LIN {X 0,Y 114.855,Z 265.173,A -85,B 0,C 180,E1 -25888.942,E2 -25888.942} C_VEL
LIN {X 0,Y 114.946,Z 265.116,A -85,B 0,C 180,E1 -25896.507,E2 -25896.507} C_VEL
LIN {X 0,Y 115.013,Z 265.157,A -85,B 0,C 180,E1 -25902.21,E2 -25902.21} C_VEL
LIN {X 0,Y 115.285,Z 265.077,A -85,B 0,C 180,E1 -25907.258,E2 -25907.258} C_VEL
LIN {X 0,Y 115.397,Z 265.09,A -85,B 0,C 180,E1 -25913.003,E2 -25913.003} C_VEL
LIN {X 0,Y 115.994,Z 264.995,A -85,B 0,C 180,E1 -25920,E2 -25920} C_VEL
LIN {X 0,Y 115.392,Z 265.108,A -85,B 0,C 180,E1 -25926.996,E2 -25926.996} C_VEL
LIN {X 0,Y 115.284,Z 265.085,A -85,B 0,C 180,E1 -25932.739,E2 -25932.739} C_VEL
LIN {X 0,Y 114.998,Z 265.157,A -85,B 0,C 180,E1 -25939.525,E2 -25939.525} C_VEL
LIN {X 0,Y 115.938,Z 267.926,A -85,B 0,C 180,E1 -25940.747,E2 -25940.747} C_VEL
LIN {X 0,Y 117.848,Z 270.02,A -85,B 0,C 180,E1 -25942.524,E2 -25942.524} C_VEL
LIN {X 0,Y 119.053,Z 270.961,A -85,B 0,C 180,E1 -25943.531,E2 -25943.531} C_VEL
LIN {X 0,Y 120.863,Z 274.022,A -85,B 0,C 180,E1 -25945.164,E2 -25945.164} C_VEL
LIN {X 0,Y 122.793,Z 276.078,A -85,B 0,C 180,E1 -25946.675,E2 -25946.675} C_VEL
LIN {X 0,Y 125.302,Z 279.71,A -85,B 0,C 180,E1 -25948.59,E2 -25948.59} C_VEL
LIN {X 0,Y 129.507,Z 285.851,A -85,B 0,C 180,E1 -25951.488,E2 -25951.488} C_VEL
LIN {X 0,Y 134.666,Z 293.955,A -85,B 0,C 180,E1 -25954.693,E2 -25954.693} C_VEL
LIN {X 0,Y 138.207,Z 301.272,A -85,B 0,C 180,E1 -25956.805,E2 -25956.805} C_VEL
LIN {X 0,Y 143.082,Z 312.975,A -85,B 0,C 180,E1 -25959.569,E2 -25959.569} C_VEL
LIN {X 0,Y 147.64,Z 326.29,A -85,B 0,C 180,E1 -25962.08,E2 -25962.08} C_VEL
LIN {X 0,Y 144.395,Z 368.364,A -85,B 0,C 180,E1 -25963.988,E2 -25963.988} C_VEL
LIN {X 0,Y 142.249,Z 381.813,A -85,B 0,C 180,E1 -25965.008,E2 -25965.008} C_VEL
LIN {X 0,Y 139.648,Z 394.07,A -85,B 0,C 180,E1 -25966.462,E2 -25966.462} C_VEL
LIN {X 0,Y 136.244,Z 405.888,A -85,B 0,C 180,E1 -25968.385,E2 -25968.385} C_VEL
LIN {X 0,Y 132.886,Z 416.032,A -85,B 0,C 180,E1 -25970.607,E2 -25970.607} C_VEL
LIN {X 0,Y 128.827,Z 426.583,A -85,B 0,C 180,E1 -25973.611,E2 -25973.611} C_VEL
LIN {X 0,Y 125.2,Z 435.221,A -85,B 0,C 180,E1 -25976.819,E2 -25976.819} C_VEL
LIN {X 0,Y 121.652,Z 443.346,A -85,B 0,C 180,E1 -25980.697,E2 -25980.697} C_VEL
LIN {X 0,Y 118.219,Z 450.929,A -85,B 0,C 180,E1 -25985.41,E2 -25985.41} C_VEL
LIN {X 0,Y 115.387,Z 457.118,A -85,B 0,C 180,E1 -25990.429,E2 -25990.429} C_VEL
LIN {X 0,Y 113.579,Z 462.024,A -85,B 0,C 180,E1 -25995.67,E2 -25995.67} C_VEL
LIN {X 0,Y 112.543,Z 465.767,A -85,B 0,C 180,E1 -26001.019,E2 -26001.019} C_VEL
LIN {X 0,Y 112.201,Z 468.455,A -85,B 0,C 180,E1 -26006.409,E2 -26006.409} C_VEL
LIN {X 0,Y 112.263,Z 469.704,A -85,B 0,C 180,E1 -26010.001,E2 -26010.001} C_VEL
LIN {X 0,Y 112.2,Z 470.534,A -85,B 0,C 180,E1 -26013.592,E2 -26013.592} C_VEL
LIN {X 0,Y 112.334,Z 470.932,A -85,B 0,C 180,E1 -26017.189,E2 -26017.189} C_VEL
LIN {X 0,Y 113.649,Z 470.568,A -85,B 0,C 180,E1 -26024.322,E2 -26024.322} C_VEL
LIN {X 0,Y 116.47,Z 468.695,A -85,B 0,C 180,E1 -26031.227,E2 -26031.227} C_VEL
LIN {X 0,Y 121.115,Z 465.171,A -85,B 0,C 180,E1 -26037.66,E2 -26037.66} C_VEL
LIN {X 0,Y 125.472,Z 461.407,A -85,B 0,C 180,E1 -26042.149,E2 -26042.149} C_VEL
LIN {X 0,Y 130.501,Z 456.57,A -85,B 0,C 180,E1 -26046.327,E2 -26046.327} C_VEL
LIN {X 0,Y 137.171,Z 449.407,A -85,B 0,C 180,E1 -26050.787,E2 -26050.787} C_VEL
LIN {X 0,Y 143.707,Z 441.626,A -85,B 0,C 180,E1 -26054.179,E2 -26054.179} C_VEL
LIN {X 0,Y 150.624,Z 432.012,A -85,B 0,C 180,E1 -26057.298,E2 -26057.298} C_VEL
LIN {X 0,Y 156.829,Z 422.095,A -85,B 0,C 180,E1 -26059.625,E2 -26059.625} C_VEL
LIN {X 0,Y 159.223,Z 417.796,A -85,B 0,C 180,E1 -26060.431,E2 -26060.431} C_VEL
LIN {X 0,Y 161.357,Z 413.071,A -85,B 0,C 180,E1 -26061.461,E2 -26061.461} C_VEL
LIN {X 0,Y 163.563,Z 405.279,A -85,B 0,C 180,E1 -26063.505,E2 -26063.505} C_VEL
LIN {X 0,Y 165.482,Z 397.087,A -85,B 0,C 180,E1 -26065.314,E2 -26065.314} C_VEL
LIN {X 0,Y 167.06,Z 391.752,A -85,B 0,C 180,E1 -26065.968,E2 -26065.968} C_VEL
LIN {X 0,Y 170.943,Z 378.184,A -85,B 0,C 180,E1 -26066.933,E2 -26066.933} C_VEL
LIN {X 0,Y 173.358,Z 365.954,A -85,B 0,C 180,E1 -26067.492,E2 -26067.492} C_VEL
LIN {X 0,Y 175.241,Z 348.208,A -85,B 0,C 180,E1 -26068.166,E2 -26068.166} C_VEL
LIN {X 0,Y 173.221,Z 341.92,A -85,B 0,C 180,E1 -26070.659,E2 -26070.659} C_VEL
LIN {X 0,Y 171.373,Z 336.851,A -85,B 0,C 180,E1 -26073.277,E2 -26073.277} C_VEL
LIN {X 0,Y 169.812,Z 332.855,A -85,B 0,C 180,E1 -26075.909,E2 -26075.909} C_VEL
LIN {X 0,Y 168.758,Z 330.738,A -85,B 0,C 180,E1 -26077.988,E2 -26077.988} C_VEL
LIN {X 0,Y 167.065,Z 326.954,A -85,B 0,C 180,E1 -26083.227,E2 -26083.227} C_VEL
LIN {X 0,Y 166.739,Z 326.515,A -85,B 0,C 180,E1 -26090.294,E2 -26090.294} C_VEL
LIN {X 0,Y 167.542,Z 327.166,A -85,B 0,C 180,E1 -26093.868,E2 -26093.868} C_VEL
LIN {X 0,Y 169.247,Z 331.048,A -85,B 0,C 180,E1 -26098.353,E2 -26098.353} C_VEL
LIN {X 0,Y 171.178,Z 334.972,A -85,B 0,C 180,E1 -26101.648,E2 -26101.648} C_VEL
LIN {X 0,Y 173.938,Z 340.804,A -85,B 0,C 180,E1 -26105.301,E2 -26105.301} C_VEL
LIN {X 0,Y 175.586,Z 344.85,A -85,B 0,C 180,E1 -26107.174,E2 -26107.174} C_VEL
LIN {X 0,Y 173.207,Z 364.688,A -85,B 0,C 180,E1 -26107.837,E2 -26107.837} C_VEL
LIN {X 0,Y 170.577,Z 377.505,A -85,B 0,C 180,E1 -26108.571,E2 -26108.571} C_VEL
LIN {X 0,Y 166.926,Z 389.808,A -85,B 0,C 180,E1 -26109.597,E2 -26109.597} C_VEL
LIN {X 0,Y 162.787,Z 400.561,A -85,B 0,C 180,E1 -26110.831,E2 -26110.831} C_VEL
LIN {X 0,Y 157.521,Z 411.598,A -85,B 0,C 180,E1 -26112.516,E2 -26112.516} C_VEL
LIN {X 0,Y 151.614,Z 421.914,A -85,B 0,C 180,E1 -26114.614,E2 -26114.614} C_VEL
LIN {X 0,Y 145.495,Z 430.892,A -85,B 0,C 180,E1 -26117.028,E2 -26117.028} C_VEL
LIN {X 0,Y 138.67,Z 439.441,A -85,B 0,C 180,E1 -26120.118,E2 -26120.118} C_VEL
LIN {X 0,Y 132.225,Z 446.432,A -85,B 0,C 180,E1 -26123.528,E2 -26123.528} C_VEL
LIN {X 0,Y 126.447,Z 451.978,A -85,B 0,C 180,E1 -26127.216,E2 -26127.216} C_VEL
LIN {X 0,Y 120.926,Z 456.69,A -85,B 0,C 180,E1 -26131.538,E2 -26131.538} C_VEL
LIN {X 0,Y 114.755,Z 461.213,A -85,B 0,C 180,E1 -26137.766,E2 -26137.766} C_VEL
LIN {X 0,Y 110.03,Z 464.019,A -85,B 0,C 180,E1 -26144.637,E2 -26144.637} C_VEL
LIN {X 0,Y 106.69,Z 465.22,A -85,B 0,C 180,E1 -26152.231,E2 -26152.231} C_VEL
LIN {X 0,Y 105.248,Z 465.079,A -85,B 0,C 180,E1 -26157.71,E2 -26157.71} C_VEL
LIN {X 0,Y 104.725,Z 464.378,A -85,B 0,C 180,E1 -26161.981,E2 -26161.981} C_VEL
LIN {X 0,Y 104.598,Z 463.238,A -85,B 0,C 180,E1 -26166.225,E2 -26166.225} C_VEL
LIN {X 0,Y 105.233,Z 460.602,A -85,B 0,C 180,E1 -26172.51,E2 -26172.51} C_VEL
LIN {X 0,Y 106.709,Z 456.837,A -85,B 0,C 180,E1 -26178.604,E2 -26178.604} C_VEL
LIN {X 0,Y 108.848,Z 451.866,A -85,B 0,C 180,E1 -26184.442,E2 -26184.442} C_VEL
LIN {X 0,Y 111.866,Z 445.532,A -85,B 0,C 180,E1 -26189.999,E2 -26189.999} C_VEL
LIN {X 0,Y 115.781,Z 437.599,A -85,B 0,C 180,E1 -26195.224,E2 -26195.224} C_VEL
LIN {X 0,Y 119.644,Z 429.439,A -85,B 0,C 180,E1 -26199.296,E2 -26199.296} C_VEL
LIN {X 0,Y 123.956,Z 419.414,A -85,B 0,C 180,E1 -26203.108,E2 -26203.108} C_VEL
LIN {X 0,Y 128.326,Z 408.2,A -85,B 0,C 180,E1 -26206.3,E2 -26206.3} C_VEL
LIN {X 0,Y 131.878,Z 397.261,A -85,B 0,C 180,E1 -26208.647,E2 -26208.647} C_VEL
LIN {X 0,Y 135.122,Z 385.083,A -85,B 0,C 180,E1 -26210.573,E2 -26210.573} C_VEL
LIN {X 0,Y 137.623,Z 372.215,A -85,B 0,C 180,E1 -26212.056,E2 -26212.056} C_VEL
LIN {X 0,Y 139.422,Z 359.052,A -85,B 0,C 180,E1 -26212.988,E2 -26212.988} C_VEL
LIN {X 0,Y 142.507,Z 321.432,A -85,B 0,C 180,E1 -26214.64,E2 -26214.64} C_VEL
LIN {X 0,Y 135.741,Z 307.538,A -85,B 0,C 180,E1 -26218.335,E2 -26218.335} C_VEL
LIN {X 0,Y 130.296,Z 297.995,A -85,B 0,C 180,E1 -26221.645,E2 -26221.645} C_VEL
LIN {X 0,Y 126.382,Z 291.705,A -85,B 0,C 180,E1 -26224.24,E2 -26224.24} C_VEL
LIN {X 0,Y 121.795,Z 284.959,A -85,B 0,C 180,E1 -26227.641,E2 -26227.641} C_VEL
LIN {X 0,Y 119.203,Z 281.373,A -85,B 0,C 180,E1 -26229.767,E2 -26229.767} C_VEL
LIN {X 0,Y 116.629,Z 278.048,A -85,B 0,C 180,E1 -26232.044,E2 -26232.044} C_VEL
LIN {X 0,Y 115.814,Z 276.758,A -85,B 0,C 180,E1 -26232.844,E2 -26232.844} C_VEL
LIN {X 0,Y 113.43,Z 274.3,A -85,B 0,C 180,E1 -26235.187,E2 -26235.187} C_VEL
LIN {X 0,Y 112.045,Z 271.721,A -85,B 0,C 180,E1 -26236.838,E2 -26236.838} C_VEL
LIN {X 0,Y 109.395,Z 269.857,A -85,B 0,C 180,E1 -26239.838,E2 -26239.838} C_VEL
LIN {X 0,Y 108.067,Z 267.583,A -85,B 0,C 180,E1 -26241.77,E2 -26241.77} C_VEL
LIN {X 0,Y 107.736,Z 266.027,A -85,B 0,C 180,E1 -26242.558,E2 -26242.558} C_VEL
LIN {X 0,Y 107.791,Z 266.049,A -85,B 0,C 180,E1 -26248.56,E2 -26248.56} C_VEL
LIN {X 0,Y 107.911,Z 265.992,A -85,B 0,C 180,E1 -26256.997,E2 -26256.997} C_VEL
LIN {X 0,Y 108.037,Z 266.005,A -85,B 0,C 180,E1 -26264.917,E2 -26264.917} C_VEL
LIN {X 0,Y 108.292,Z 265.939,A -85,B 0,C 180,E1 -26268.773,E2 -26268.773} C_VEL
LIN {X 0,Y 108.462,Z 265.973,A -85,B 0,C 180,E1 -26276.285,E2 -26276.285} C_VEL
LIN {X 0,Y 108.945,Z 265.871,A -85,B 0,C 180,E1 -26280,E2 -26280} C_VEL
LIN {X 0,Y 108.332,Z 265.99,A -85,B 0,C 180,E1 -26287.455,E2 -26287.455} C_VEL
LIN {X 0,Y 108.247,Z 266.109,A -85,B 0,C 180,E1 -26292.785,E2 -26292.785} C_VEL
LIN {X 0,Y 108.897,Z 268.457,A -85,B 0,C 180,E1 -26293.955,E2 -26293.955} C_VEL
LIN {X 0,Y 110.561,Z 270.663,A -85,B 0,C 180,E1 -26296.147,E2 -26296.147} C_VEL
LIN {X 0,Y 112.445,Z 271.954,A -85,B 0,C 180,E1 -26298.21,E2 -26298.21} C_VEL
LIN {X 0,Y 114.23,Z 275.148,A -85,B 0,C 180,E1 -26300.247,E2 -26300.247} C_VEL
LIN {X 0,Y 116.341,Z 277.205,A -85,B 0,C 180,E1 -26302.237,E2 -26302.237} C_VEL
LIN {X 0,Y 118.784,Z 280.769,A -85,B 0,C 180,E1 -26304.466,E2 -26304.466} C_VEL
LIN {X 0,Y 120.022,Z 282.345,A -85,B 0,C 180,E1 -26305.512,E2 -26305.512} C_VEL
LIN {X 0,Y 123.658,Z 287.644,A -85,B 0,C 180,E1 -26308.407,E2 -26308.407} C_VEL
LIN {X 0,Y 129.7,Z 297.014,A -85,B 0,C 180,E1 -26312.58,E2 -26312.58} C_VEL
LIN {X 0,Y 132.747,Z 303.036,A -85,B 0,C 180,E1 -26314.575,E2 -26314.575} C_VEL
LIN {X 0,Y 137.566,Z 314.647,A -85,B 0,C 180,E1 -26317.58,E2 -26317.58} C_VEL
LIN {X 0,Y 141.936,Z 327.343,A -85,B 0,C 180,E1 -26320.19,E2 -26320.19} C_VEL
LIN {X 0,Y 142.161,Z 329.138,A -85,B 0,C 180,E1 -26320.4,E2 -26320.4} C_VEL
LIN {X 0,Y 138.898,Z 368.246,A -85,B 0,C 180,E1 -26322.179,E2 -26322.179} C_VEL
LIN {X 0,Y 136.583,Z 382.144,A -85,B 0,C 180,E1 -26323.257,E2 -26323.257} C_VEL
LIN {X 0,Y 133.695,Z 394.706,A -85,B 0,C 180,E1 -26324.794,E2 -26324.794} C_VEL
LIN {X 0,Y 129.98,Z 407.17,A -85,B 0,C 180,E1 -26326.951,E2 -26326.951} C_VEL
LIN {X 0,Y 125.98,Z 418.334,A -85,B 0,C 180,E1 -26329.571,E2 -26329.571} C_VEL
LIN {X 0,Y 121.817,Z 428.374,A -85,B 0,C 180,E1 -26332.716,E2 -26332.716} C_VEL
LIN {X 0,Y 117.714,Z 437.49,A -85,B 0,C 180,E1 -26336.479,E2 -26336.479} C_VEL
LIN {X 0,Y 114.269,Z 445.026,A -85,B 0,C 180,E1 -26340.527,E2 -26340.527} C_VEL
LIN {X 0,Y 110.649,Z 452.386,A -85,B 0,C 180,E1 -26345.617,E2 -26345.617} C_VEL
LIN {X 0,Y 107.874,Z 458.258,A -85,B 0,C 180,E1 -26350.99,E2 -26350.99} C_VEL
LIN {X 0,Y 106.202,Z 462.871,A -85,B 0,C 180,E1 -26356.609,E2 -26356.609} C_VEL
LIN {X 0,Y 105.293,Z 466.345,A -85,B 0,C 180,E1 -26362.329,E2 -26362.329} C_VEL
LIN {X 0,Y 105.111,Z 468.063,A -85,B 0,C 180,E1 -26366.167,E2 -26366.167} C_VEL
LIN {X 0,Y 105.175,Z 469.355,A -85,B 0,C 180,E1 -26370.001,E2 -26370.001} C_VEL
LIN {X 0,Y 105.11,Z 470.227,A -85,B 0,C 180,E1 -26373.834,E2 -26373.834} C_VEL
LIN {X 0,Y 105.277,Z 470.704,A -85,B 0,C 180,E1 -26377.673,E2 -26377.673} C_VEL
LIN {X 0,Y 106.758,Z 470.439,A -85,B 0,C 180,E1 -26385.268,E2 -26385.268} C_VEL
LIN {X 0,Y 109.863,Z 468.676,A -85,B 0,C 180,E1 -26392.571,E2 -26392.571} C_VEL
LIN {X 0,Y 112.168,Z 467.196,A -85,B 0,C 180,E1 -26396.014,E2 -26396.014} C_VEL
LIN {X 0,Y 117.847,Z 462.955,A -85,B 0,C 180,E1 -26402.462,E2 -26402.462} C_VEL
LIN {X 0,Y 123.207,Z 458.44,A -85,B 0,C 180,E1 -26407.004,E2 -26407.004} C_VEL
LIN {X 0,Y 129.801,Z 452.116,A -85,B 0,C 180,E1 -26411.55,E2 -26411.55} C_VEL
LIN {X 0,Y 136.403,Z 445.036,A -85,B 0,C 180,E1 -26415.109,E2 -26415.109} C_VEL
LIN {X 0,Y 143.472,Z 436.291,A -85,B 0,C 180,E1 -26418.334,E2 -26418.334} C_VEL
LIN {X 0,Y 149.755,Z 427.365,A -85,B 0,C 180,E1 -26420.746,E2 -26420.746} C_VEL
LIN {X 0,Y 155.708,Z 417.573,A -85,B 0,C 180,E1 -26422.704,E2 -26422.704} C_VEL
LIN {X 0,Y 161.094,Z 406.819,A -85,B 0,C 180,E1 -26424.346,E2 -26424.346} C_VEL
LIN {X 0,Y 165.931,Z 394.934,A -85,B 0,C 180,E1 -26425.682,E2 -26425.682} C_VEL
LIN {X 0,Y 167.06,Z 391.752,A -85,B 0,C 180,E1 -26425.968,E2 -26425.968} C_VEL
LIN {X 0,Y 167.991,Z 388.123,A -85,B 0,C 180,E1 -26426.448,E2 -26426.448} C_VEL
LIN {X 0,Y 168.439,Z 382.548,A -85,B 0,C 180,E1 -26427.759,E2 -26427.759} C_VEL
LIN {X 0,Y 168.77,Z 376.886,A -85,B 0,C 180,E1 -26429.01,E2 -26429.01} C_VEL
LIN {X 0,Y 169.349,Z 373.126,A -85,B 0,C 180,E1 -26429.401,E2 -26429.401} C_VEL
LIN {X 0,Y 171.472,Z 359.966,A -85,B 0,C 180,E1 -26429.912,E2 -26429.912} C_VEL
LIN {X 0,Y 172.331,Z 351.573,A -85,B 0,C 180,E1 -26430.218,E2 -26430.218} C_VEL
LIN {X 0,Y 170.483,Z 345.518,A -85,B 0,C 180,E1 -26432.914,E2 -26432.914} C_VEL
LIN {X 0,Y 169.288,Z 342.061,A -85,B 0,C 180,E1 -26434.914,E2 -26434.914} C_VEL
LIN {X 0,Y 168.233,Z 339.129,A -85,B 0,C 180,E1 -26436.939,E2 -26436.939} C_VEL
LIN {X 0,Y 167.536,Z 337.541,A -85,B 0,C 180,E1 -26438.516,E2 -26438.516} C_VEL
LIN {X 0,Y 166.05,Z 333.957,A -85,B 0,C 180,E1 -26443.526,E2 -26443.526} C_VEL
LIN {X 0,Y 165.784,Z 333.552,A -85,B 0,C 180,E1 -26450.237,E2 -26450.237} C_VEL
LIN {X 0,Y 166.447,Z 334.154,A -85,B 0,C 180,E1 -26453.46,E2 -26453.46} C_VEL
LIN {X 0,Y 167.891,Z 337.672,A -85,B 0,C 180,E1 -26457.601,E2 -26457.601} C_VEL
LIN {X 0,Y 169.693,Z 341.69,A -85,B 0,C 180,E1 -26460.987,E2 -26460.987} C_VEL
LIN {X 0,Y 172.062,Z 347.151,A -85,B 0,C 180,E1 -26464.415,E2 -26464.415} C_VEL
LIN {X 0,Y 172.599,Z 348.504,A -85,B 0,C 180,E1 -26465.088,E2 -26465.088} C_VEL
LIN {X 0,Y 170.388,Z 365.81,A -85,B 0,C 180,E1 -26465.685,E2 -26465.685} C_VEL
LIN {X 0,Y 167.678,Z 378.305,A -85,B 0,C 180,E1 -26466.391,E2 -26466.391} C_VEL
LIN {X 0,Y 163.89,Z 390.477,A -85,B 0,C 180,E1 -26467.392,E2 -26467.392} C_VEL
LIN {X 0,Y 159.096,Z 402.269,A -85,B 0,C 180,E1 -26468.733,E2 -26468.733} C_VEL
LIN {X 0,Y 153.375,Z 413.542,A -85,B 0,C 180,E1 -26470.468,E2 -26470.468} C_VEL
LIN {X 0,Y 146.789,Z 424.13,A -85,B 0,C 180,E1 -26472.705,E2 -26472.705} C_VEL
LIN {X 0,Y 139.888,Z 433.388,A -85,B 0,C 180,E1 -26475.302,E2 -26475.302} C_VEL
LIN {X 0,Y 132.679,Z 441.713,A -85,B 0,C 180,E1 -26478.532,E2 -26478.532} C_VEL
LIN {X 0,Y 125.538,Z 448.723,A -85,B 0,C 180,E1 -26482.29,E2 -26482.29} C_VEL
LIN {X 0,Y 118.349,Z 454.861,A -85,B 0,C 180,E1 -26487.032,E2 -26487.032} C_VEL
LIN {X 0,Y 112.152,Z 459.405,A -85,B 0,C 180,E1 -26492.223,E2 -26492.223} C_VEL
LIN {X 0,Y 106.95,Z 462.602,A -85,B 0,C 180,E1 -26497.949,E2 -26497.949} C_VEL
LIN {X 0,Y 103.79,Z 464.201,A -85,B 0,C 180,E1 -26502.621,E2 -26502.621} C_VEL
LIN {X 0,Y 101.771,Z 465.003,A -85,B 0,C 180,E1 -26506.324,E2 -26506.324} C_VEL
LIN {X 0,Y 99.987,Z 465.424,A -85,B 0,C 180,E1 -26510.757,E2 -26510.757} C_VEL
LIN {X 0,Y 98.621,Z 465.374,A -85,B 0,C 180,E1 -26515.242,E2 -26515.242} C_VEL
LIN {X 0,Y 97.823,Z 464.854,A -85,B 0,C 180,E1 -26519.807,E2 -26519.807} C_VEL
LIN {X 0,Y 97.484,Z 463.815,A -85,B 0,C 180,E1 -26524.369,E2 -26524.369} C_VEL
LIN {X 0,Y 97.675,Z 462.187,A -85,B 0,C 180,E1 -26529.293,E2 -26529.293} C_VEL
LIN {X 0,Y 98.719,Z 459.164,A -85,B 0,C 180,E1 -26535.571,E2 -26535.571} C_VEL
LIN {X 0,Y 100.589,Z 454.847,A -85,B 0,C 180,E1 -26541.967,E2 -26541.967} C_VEL
LIN {X 0,Y 103.855,Z 448.173,A -85,B 0,C 180,E1 -26549.03,E2 -26549.03} C_VEL
LIN {X 0,Y 107.638,Z 440.878,A -85,B 0,C 180,E1 -26554.681,E2 -26554.681} C_VEL
LIN {X 0,Y 111.463,Z 433.363,A -85,B 0,C 180,E1 -26559.069,E2 -26559.069} C_VEL
LIN {X 0,Y 116.196,Z 423.347,A -85,B 0,C 180,E1 -26563.482,E2 -26563.482} C_VEL
LIN {X 0,Y 120.699,Z 412.866,A -85,B 0,C 180,E1 -26566.925,E2 -26566.925} C_VEL
LIN {X 0,Y 124.894,Z 401.356,A -85,B 0,C 180,E1 -26569.732,E2 -26569.732} C_VEL
LIN {X 0,Y 128.666,Z 388.814,A -85,B 0,C 180,E1 -26571.975,E2 -26571.975} C_VEL
LIN {X 0,Y 131.513,Z 376.169,A -85,B 0,C 180,E1 -26573.596,E2 -26573.596} C_VEL
LIN {X 0,Y 133.596,Z 363.212,A -85,B 0,C 180,E1 -26574.686,E2 -26574.686} C_VEL
LIN {X 0,Y 136.055,Z 336.575,A -85,B 0,C 180,E1 -26575.937,E2 -26575.937} C_VEL
LIN {X 0,Y 137.102,Z 323.784,A -85,B 0,C 180,E1 -26576.505,E2 -26576.505} C_VEL
LIN {X 0,Y 130.752,Z 310.493,A -85,B 0,C 180,E1 -26580.331,E2 -26580.331} C_VEL
LIN {X 0,Y 123.801,Z 298.36,A -85,B 0,C 180,E1 -26585.047,E2 -26585.047} C_VEL
LIN {X 0,Y 118.6,Z 290.493,A -85,B 0,C 180,E1 -26589.163,E2 -26589.163} C_VEL
LIN {X 0,Y 116.229,Z 287.158,A -85,B 0,C 180,E1 -26591.245,E2 -26591.245} C_VEL
LIN {X 0,Y 113.609,Z 283.39,A -85,B 0,C 180,E1 -26593.806,E2 -26593.806} C_VEL
LIN {X 0,Y 110.591,Z 279.729,A -85,B 0,C 180,E1 -26597.074,E2 -26597.074} C_VEL
LIN {X 0,Y 109.653,Z 278.141,A -85,B 0,C 180,E1 -26598.251,E2 -26598.251} C_VEL
LIN {X 0,Y 107.104,Z 275.941,A -85,B 0,C 180,E1 -26601.454,E2 -26601.454} C_VEL
LIN {X 0,Y 105.682,Z 273.048,A -85,B 0,C 180,E1 -26603.828,E2 -26603.828} C_VEL
LIN {X 0,Y 104.474,Z 272.366,A -85,B 0,C 180,E1 -26605.709,E2 -26605.709} C_VEL
LIN {X 0,Y 101.662,Z 269.762,A -85,B 0,C 180,E1 -26611.341,E2 -26611.341} C_VEL
LIN {X 0,Y 100.783,Z 267.269,A -85,B 0,C 180,E1 -26614.273,E2 -26614.273} C_VEL
LIN {X 0,Y 100.737,Z 266.886,A -85,B 0,C 180,E1 -26614.758,E2 -26614.758} C_VEL
LIN {X 0,Y 100.816,Z 266.896,A -85,B 0,C 180,E1 -26619.601,E2 -26619.601} C_VEL
LIN {X 0,Y 101.19,Z 266.824,A -85,B 0,C 180,E1 -26627.973,E2 -26627.973} C_VEL
LIN {X 0,Y 101.274,Z 266.829,A -85,B 0,C 180,E1 -26632.022,E2 -26632.022} C_VEL
LIN {X 0,Y 101.869,Z 266.751,A -85,B 0,C 180,E1 -26640,E2 -26640} C_VEL
LIN {X 0,Y 101.58,Z 266.992,A -85,B 0,C 180,E1 -26642.23,E2 -26642.23} C_VEL
LIN {X 0,Y 102.128,Z 269.229,A -85,B 0,C 180,E1 -26644.069,E2 -26644.069} C_VEL
LIN {X 0,Y 103.866,Z 271.526,A -85,B 0,C 180,E1 -26647.777,E2 -26647.777} C_VEL
LIN {X 0,Y 106.045,Z 272.825,A -85,B 0,C 180,E1 -26651.226,E2 -26651.226} C_VEL
LIN {X 0,Y 107.515,Z 275.955,A -85,B 0,C 180,E1 -26653.636,E2 -26653.636} C_VEL
LIN {X 0,Y 110.202,Z 278.596,A -85,B 0,C 180,E1 -26656.991,E2 -26656.991} C_VEL
LIN {X 0,Y 112.398,Z 281.988,A -85,B 0,C 180,E1 -26659.564,E2 -26659.564} C_VEL
LIN {X 0,Y 113.853,Z 283.623,A -85,B 0,C 180,E1 -26661.041,E2 -26661.041} C_VEL
LIN {X 0,Y 117.239,Z 288.397,A -85,B 0,C 180,E1 -26664.245,E2 -26664.245} C_VEL
LIN {X 0,Y 121.876,Z 295.355,A -85,B 0,C 180,E1 -26668.111,E2 -26668.111} C_VEL
LIN {X 0,Y 127.48,Z 304.893,A -85,B 0,C 180,E1 -26672.164,E2 -26672.164} C_VEL
LIN {X 0,Y 132.436,Z 316.969,A -85,B 0,C 180,E1 -26675.597,E2 -26675.597} C_VEL
LIN {X 0,Y 136.797,Z 329.994,A -85,B 0,C 180,E1 -26678.452,E2 -26678.452} C_VEL
LIN {X 0,Y 133.532,Z 368.108,A -85,B 0,C 180,E1 -26680.237,E2 -26680.237} C_VEL
LIN {X 0,Y 131.155,Z 381.776,A -85,B 0,C 180,E1 -26681.3,E2 -26681.3} C_VEL
LIN {X 0,Y 128.211,Z 394.27,A -85,B 0,C 180,E1 -26682.849,E2 -26682.849} C_VEL
LIN {X 0,Y 124.308,Z 406.769,A -85,B 0,C 180,E1 -26685.033,E2 -26685.033} C_VEL
LIN {X 0,Y 120.122,Z 417.972,A -85,B 0,C 180,E1 -26687.715,E2 -26687.715} C_VEL
LIN {X 0,Y 116.229,Z 427.049,A -85,B 0,C 180,E1 -26690.588,E2 -26690.588} C_VEL
LIN {X 0,Y 111.807,Z 436.356,A -85,B 0,C 180,E1 -26694.449,E2 -26694.449} C_VEL
LIN {X 0,Y 108.057,Z 444.044,A -85,B 0,C 180,E1 -26698.647,E2 -26698.647} C_VEL
LIN {X 0,Y 104.195,Z 451.547,A -85,B 0,C 180,E1 -26703.997,E2 -26703.997} C_VEL
LIN {X 0,Y 101.153,Z 457.541,A -85,B 0,C 180,E1 -26709.673,E2 -26709.673} C_VEL
LIN {X 0,Y 99.263,Z 462.27,A -85,B 0,C 180,E1 -26715.653,E2 -26715.653} C_VEL
LIN {X 0,Y 98.262,Z 465.845,A -85,B 0,C 180,E1 -26721.777,E2 -26721.777} C_VEL
LIN {X 0,Y 98.022,Z 467.653,A -85,B 0,C 180,E1 -26725.889,E2 -26725.889} C_VEL
LIN {X 0,Y 98.08,Z 468.993,A -85,B 0,C 180,E1 -26730.001,E2 -26730.001} C_VEL
LIN {X 0,Y 98.02,Z 469.912,A -85,B 0,C 180,E1 -26734.112,E2 -26734.112} C_VEL
LIN {X 0,Y 98.245,Z 470.443,A -85,B 0,C 180,E1 -26738.226,E2 -26738.226} C_VEL
LIN {X 0,Y 98.828,Z 470.583,A -85,B 0,C 180,E1 -26742.319,E2 -26742.319} C_VEL
LIN {X 0,Y 101.36,Z 469.663,A -85,B 0,C 180,E1 -26750.285,E2 -26750.285} C_VEL
LIN {X 0,Y 105.824,Z 467.246,A -85,B 0,C 180,E1 -26757.703,E2 -26757.703} C_VEL
LIN {X 0,Y 110.248,Z 464.34,A -85,B 0,C 180,E1 -26762.81,E2 -26762.81} C_VEL
LIN {X 0,Y 115.543,Z 460.451,A -85,B 0,C 180,E1 -26767.464,E2 -26767.464} C_VEL
LIN {X 0,Y 121.381,Z 455.492,A -85,B 0,C 180,E1 -26771.748,E2 -26771.748} C_VEL
LIN {X 0,Y 127.955,Z 449.303,A -85,B 0,C 180,E1 -26775.564,E2 -26775.564} C_VEL
LIN {X 0,Y 135.219,Z 441.613,A -85,B 0,C 180,E1 -26778.907,E2 -26778.907} C_VEL
LIN {X 0,Y 141.46,Z 433.863,A -85,B 0,C 180,E1 -26781.489,E2 -26781.489} C_VEL
LIN {X 0,Y 147.461,Z 425.481,A -85,B 0,C 180,E1 -26783.539,E2 -26783.539} C_VEL
LIN {X 0,Y 154.332,Z 414.039,A -85,B 0,C 180,E1 -26785.627,E2 -26785.627} C_VEL
LIN {X 0,Y 159.967,Z 402.535,A -85,B 0,C 180,E1 -26787.165,E2 -26787.165} C_VEL
LIN {X 0,Y 164.648,Z 390.37,A -85,B 0,C 180,E1 -26788.324,E2 -26788.324} C_VEL
LIN {X 0,Y 168.507,Z 376.996,A -85,B 0,C 180,E1 -26789.206,E2 -26789.206} C_VEL
LIN {X 0,Y 169.349,Z 373.126,A -85,B 0,C 180,E1 -26789.401,E2 -26789.401} C_VEL
LIN {X 0,Y 170.185,Z 367.824,A -85,B 0,C 180,E1 -26789.777,E2 -26789.777} C_VEL
LIN {X 0,Y 170.397,Z 362.735,A -85,B 0,C 180,E1 -26790.467,E2 -26790.467} C_VEL
LIN {X 0,Y 170.106,Z 358.107,A -85,B 0,C 180,E1 -26791.447,E2 -26791.447} C_VEL
LIN {X 0,Y 169.435,Z 354.226,A -85,B 0,C 180,E1 -26792.723,E2 -26792.723} C_VEL
LIN {X 0,Y 167.844,Z 348.806,A -85,B 0,C 180,E1 -26795.587,E2 -26795.587} C_VEL
LIN {X 0,Y 166.741,Z 345.381,A -85,B 0,C 180,E1 -26798.015,E2 -26798.015} C_VEL
LIN {X 0,Y 166.216,Z 344.24,A -85,B 0,C 180,E1 -26799.311,E2 -26799.311} C_VEL
LIN {X 0,Y 164.973,Z 340.911,A -85,B 0,C 180,E1 -26804.178,E2 -26804.178} C_VEL
LIN {X 0,Y 164.937,Z 340.683,A -85,B 0,C 180,E1 -26810.913,E2 -26810.913} C_VEL
LIN {X 0,Y 165.386,Z 341.184,A -85,B 0,C 180,E1 -26813.094,E2 -26813.094} C_VEL
LIN {X 0,Y 166.626,Z 344.483,A -85,B 0,C 180,E1 -26817.002,E2 -26817.002} C_VEL
LIN {X 0,Y 168.157,Z 348.196,A -85,B 0,C 180,E1 -26820.18,E2 -26820.18} C_VEL
LIN {X 0,Y 169.883,Z 352.403,A -85,B 0,C 180,E1 -26822.939,E2 -26822.939} C_VEL
LIN {X 0,Y 167.812,Z 367.205,A -85,B 0,C 180,E1 -26823.467,E2 -26823.467} C_VEL
LIN {X 0,Y 164.861,Z 379.778,A -85,B 0,C 180,E1 -26824.195,E2 -26824.195} C_VEL
LIN {X 0,Y 160.558,Z 392.612,A -85,B 0,C 180,E1 -26825.241,E2 -26825.241} C_VEL
LIN {X 0,Y 155.631,Z 403.988,A -85,B 0,C 180,E1 -26826.547,E2 -26826.547} C_VEL
LIN {X 0,Y 150.252,Z 414.019,A -85,B 0,C 180,E1 -26828.067,E2 -26828.067} C_VEL
LIN {X 0,Y 143.68,Z 424.169,A -85,B 0,C 180,E1 -26830.134,E2 -26830.134} C_VEL
LIN {X 0,Y 136.81,Z 433.097,A -85,B 0,C 180,E1 -26832.568,E2 -26832.568} C_VEL
LIN {X 0,Y 129.626,Z 441.056,A -85,B 0,C 180,E1 -26835.491,E2 -26835.491} C_VEL
LIN {X 0,Y 122.561,Z 447.794,A -85,B 0,C 180,E1 -26838.886,E2 -26838.886} C_VEL
LIN {X 0,Y 114.896,Z 454.059,A -85,B 0,C 180,E1 -26843.432,E2 -26843.432} C_VEL
LIN {X 0,Y 108.055,Z 458.834,A -85,B 0,C 180,E1 -26848.591,E2 -26848.591} C_VEL
LIN {X 0,Y 102.161,Z 462.282,A -85,B 0,C 180,E1 -26854.358,E2 -26854.358} C_VEL
LIN {X 0,Y 97.677,Z 464.397,A -85,B 0,C 180,E1 -26860.359,E2 -26860.359} C_VEL
LIN {X 0,Y 93.421,Z 465.624,A -85,B 0,C 180,E1 -26868.79,E2 -26868.79} C_VEL
LIN {X 0,Y 91.053,Z 465.244,A -85,B 0,C 180,E1 -26877.295,E2 -26877.295} C_VEL
LIN {X 0,Y 90.466,Z 464.387,A -85,B 0,C 180,E1 -26882.217,E2 -26882.217} C_VEL
LIN {X 0,Y 90.517,Z 462.48,A -85,B 0,C 180,E1 -26888.705,E2 -26888.705} C_VEL
LIN {X 0,Y 91.821,Z 458.82,A -85,B 0,C 180,E1 -26896.725,E2 -26896.725} C_VEL
LIN {X 0,Y 93.923,Z 454.319,A -85,B 0,C 180,E1 -26903.555,E2 -26903.555} C_VEL
LIN {X 0,Y 96.966,Z 448.537,A -85,B 0,C 180,E1 -26909.999,E2 -26909.999} C_VEL
LIN {X 0,Y 100.953,Z 441.284,A -85,B 0,C 180,E1 -26915.993,E2 -26915.993} C_VEL
LIN {X 0,Y 104.977,Z 433.824,A -85,B 0,C 180,E1 -26920.608,E2 -26920.608} C_VEL
LIN {X 0,Y 110.067,Z 423.691,A -85,B 0,C 180,E1 -26925.271,E2 -26925.271} C_VEL
LIN {X 0,Y 114.705,Z 413.442,A -85,B 0,C 180,E1 -26928.763,E2 -26928.763} C_VEL
LIN {X 0,Y 119.094,Z 402.058,A -85,B 0,C 180,E1 -26931.642,E2 -26931.642} C_VEL
LIN {X 0,Y 123.05,Z 389.518,A -85,B 0,C 180,E1 -26933.957,E2 -26933.957} C_VEL
LIN {X 0,Y 125.827,Z 378.143,A -85,B 0,C 180,E1 -26935.483,E2 -26935.483} C_VEL
LIN {X 0,Y 128.031,Z 365.783,A -85,B 0,C 180,E1 -26936.622,E2 -26936.622} C_VEL
LIN {X 0,Y 129.877,Z 348.484,A -85,B 0,C 180,E1 -26937.529,E2 -26937.529} C_VEL
LIN {X 0,Y 131.782,Z 326.075,A -85,B 0,C 180,E1 -26938.545,E2 -26938.545} C_VEL
LIN {X 0,Y 126.217,Z 314.246,A -85,B 0,C 180,E1 -26942.227,E2 -26942.227} C_VEL
LIN {X 0,Y 120.306,Z 303.603,A -85,B 0,C 180,E1 -26946.615,E2 -26946.615} C_VEL
LIN {X 0,Y 115.127,Z 295.463,A -85,B 0,C 180,E1 -26951.074,E2 -26951.074} C_VEL
LIN {X 0,Y 112.924,Z 292.377,A -85,B 0,C 180,E1 -26953.203,E2 -26953.203} C_VEL
LIN {X 0,Y 110.533,Z 288.891,A -85,B 0,C 180,E1 -26955.8,E2 -26955.8} C_VEL
LIN {X 0,Y 107.91,Z 285.21,A -85,B 0,C 180,E1 -26958.977,E2 -26958.977} C_VEL
LIN {X 0,Y 104.623,Z 281.467,A -85,B 0,C 180,E1 -26963.617,E2 -26963.617} C_VEL
LIN {X 0,Y 103.664,Z 279.517,A -85,B 0,C 180,E1 -26965.403,E2 -26965.403} C_VEL
LIN {X 0,Y 100.559,Z 276.964,A -85,B 0,C 180,E1 -26971.567,E2 -26971.567} C_VEL
LIN {X 0,Y 99.446,Z 274.211,A -85,B 0,C 180,E1 -26975.354,E2 -26975.354} C_VEL
LIN {X 0,Y 99.212,Z 273.814,A -85,B 0,C 180,E1 -26976.219,E2 -26976.219} C_VEL
LIN {X 0,Y 97.607,Z 272.977,A -85,B 0,C 180,E1 -26987.525,E2 -26987.525} C_VEL
LIN {X 0,Y 99.967,Z 273.625,A -85,B 0,C 180,E1 -27000.503,E2 -27000.503} C_VEL
LIN {X 0,Y 101.147,Z 276.857,A -85,B 0,C 180,E1 -27004.233,E2 -27004.233} C_VEL
LIN {X 0,Y 103.733,Z 279.227,A -85,B 0,C 180,E1 -27009.259,E2 -27009.259} C_VEL
LIN {X 0,Y 104.217,Z 279.753,A -85,B 0,C 180,E1 -27010.073,E2 -27010.073} C_VEL
LIN {X 0,Y 106.134,Z 283.116,A -85,B 0,C 180,E1 -27013.244,E2 -27013.244} C_VEL
LIN {X 0,Y 108.008,Z 285.026,A -85,B 0,C 180,E1 -27015.691,E2 -27015.691} C_VEL
LIN {X 0,Y 110.331,Z 288.487,A -85,B 0,C 180,E1 -27018.572,E2 -27018.572} C_VEL
LIN {X 0,Y 111.739,Z 290.444,A -85,B 0,C 180,E1 -27020.133,E2 -27020.133} C_VEL
LIN {X 0,Y 114.631,Z 294.692,A -85,B 0,C 180,E1 -27023.059,E2 -27023.059} C_VEL
LIN {X 0,Y 118.441,Z 300.472,A -85,B 0,C 180,E1 -27026.446,E2 -27026.446} C_VEL
LIN {X 0,Y 123.665,Z 309.808,A -85,B 0,C 180,E1 -27030.597,E2 -27030.597} C_VEL
LIN {X 0,Y 128.069,Z 321.057,A -85,B 0,C 180,E1 -27033.909,E2 -27033.909} C_VEL
LIN {X 0,Y 131.56,Z 331.901,A -85,B 0,C 180,E1 -27036.443,E2 -27036.443} C_VEL
LIN {X 0,Y 128.254,Z 368.186,A -85,B 0,C 180,E1 -27038.158,E2 -27038.158} C_VEL
LIN {X 0,Y 125.837,Z 381.538,A -85,B 0,C 180,E1 -27039.204,E2 -27039.204} C_VEL
LIN {X 0,Y 122.876,Z 393.732,A -85,B 0,C 180,E1 -27040.727,E2 -27040.727} C_VEL
LIN {X 0,Y 119.325,Z 404.699,A -85,B 0,C 180,E1 -27042.59,E2 -27042.59} C_VEL
LIN {X 0,Y 115.997,Z 413.646,A -85,B 0,C 180,E1 -27044.611,E2 -27044.611} C_VEL
LIN {X 0,Y 111.319,Z 424.52,A -85,B 0,C 180,E1 -27047.872,E2 -27047.872} C_VEL
LIN {X 0,Y 106.068,Z 435.183,A -85,B 0,C 180,E1 -27052.201,E2 -27052.201} C_VEL
LIN {X 0,Y 101.967,Z 443.036,A -85,B 0,C 180,E1 -27056.538,E2 -27056.538} C_VEL
LIN {X 0,Y 97.827,Z 450.689,A -85,B 0,C 180,E1 -27062.163,E2 -27062.163} C_VEL
LIN {X 0,Y 94.5,Z 456.809,A -85,B 0,C 180,E1 -27068.171,E2 -27068.171} C_VEL
LIN {X 0,Y 92.357,Z 461.651,A -85,B 0,C 180,E1 -27074.555,E2 -27074.555} C_VEL
LIN {X 0,Y 91.227,Z 465.335,A -85,B 0,C 180,E1 -27081.137,E2 -27081.137} C_VEL
LIN {X 0,Y 90.931,Z 467.218,A -85,B 0,C 180,E1 -27085.568,E2 -27085.568} C_VEL
LIN {X 0,Y 90.996,Z 468.632,A -85,B 0,C 180,E1 -27090.001,E2 -27090.001} C_VEL
LIN {X 0,Y 90.929,Z 469.597,A -85,B 0,C 180,E1 -27094.434,E2 -27094.434} C_VEL
LIN {X 0,Y 91.211,Z 470.174,A -85,B 0,C 180,E1 -27098.866,E2 -27098.866} C_VEL
LIN {X 0,Y 93.061,Z 470.184,A -85,B 0,C 180,E1 -27107.583,E2 -27107.583} C_VEL
LIN {X 0,Y 96.883,Z 468.624,A -85,B 0,C 180,E1 -27115.802,E2 -27115.802} C_VEL
LIN {X 0,Y 102.653,Z 465.541,A -85,B 0,C 180,E1 -27123.21,E2 -27123.21} C_VEL
LIN {X 0,Y 108.06,Z 462.094,A -85,B 0,C 180,E1 -27128.161,E2 -27128.161} C_VEL
LIN {X 0,Y 114.036,Z 457.622,A -85,B 0,C 180,E1 -27132.682,E2 -27132.682} C_VEL
LIN {X 0,Y 121.906,Z 450.946,A -85,B 0,C 180,E1 -27137.312,E2 -27137.312} C_VEL
LIN {X 0,Y 129.375,Z 443.716,A -85,B 0,C 180,E1 -27140.724,E2 -27140.724} C_VEL
LIN {X 0,Y 137.19,Z 434.82,A -85,B 0,C 180,E1 -27143.789,E2 -27143.789} C_VEL
LIN {X 0,Y 144.105,Z 425.67,A -85,B 0,C 180,E1 -27146.006,E2 -27146.006} C_VEL
LIN {X 0,Y 151.211,Z 414.306,A -85,B 0,C 180,E1 -27148.019,E2 -27148.019} C_VEL
LIN {X 0,Y 157.022,Z 402.925,A -85,B 0,C 180,E1 -27149.496,E2 -27149.496} C_VEL
LIN {X 0,Y 161.466,Z 392.054,A -85,B 0,C 180,E1 -27150.52,E2 -27150.52} C_VEL
LIN {X 0,Y 165.495,Z 379.094,A -85,B 0,C 180,E1 -27151.376,E2 -27151.376} C_VEL
LIN {X 0,Y 168.257,Z 366.253,A -85,B 0,C 180,E1 -27151.939,E2 -27151.939} C_VEL
LIN {X 0,Y 169.644,Z 355.075,A -85,B 0,C 180,E1 -27152.365,E2 -27152.365} C_VEL
LIN {X 0,Y 169.435,Z 354.226,A -85,B 0,C 180,E1 -27152.723,E2 -27152.723} C_VEL
LIN {X 0,Y 168.695,Z 352.421,A -85,B 0,C 180,E1 -27153.869,E2 -27153.869} C_VEL
LIN {X 0,Y 167.796,Z 351.595,A -85,B 0,C 180,E1 -27155.154,E2 -27155.154} C_VEL
LIN {X 0,Y 165.055,Z 351.1,A -85,B 0,C 180,E1 -27159.789,E2 -27159.789} C_VEL
LIN {X 0,Y 164.003,Z 347.936,A -85,B 0,C 180,E1 -27164.305,E2 -27164.305} C_VEL
LIN {X 0,Y 163.919,Z 347.651,A -85,B 0,C 180,E1 -27170.442,E2 -27170.442} C_VEL
LIN {X 0,Y 164.322,Z 348.107,A -85,B 0,C 180,E1 -27172.628,E2 -27172.628} C_VEL
LIN {X 0,Y 165.419,Z 351.376,A -85,B 0,C 180,E1 -27176.493,E2 -27176.493} C_VEL
LIN {X 0,Y 166.711,Z 354.882,A -85,B 0,C 180,E1 -27179.472,E2 -27179.472} C_VEL
LIN {X 0,Y 167.414,Z 357.007,A -85,B 0,C 180,E1 -27180.8,E2 -27180.8} C_VEL
LIN {X 0,Y 165.161,Z 370.272,A -85,B 0,C 180,E1 -27181.274,E2 -27181.274} C_VEL
LIN {X 0,Y 161.745,Z 383.156,A -85,B 0,C 180,E1 -27182.027,E2 -27182.027} C_VEL
LIN {X 0,Y 157.547,Z 394.696,A -85,B 0,C 180,E1 -27182.983,E2 -27182.983} C_VEL
LIN {X 0,Y 152.401,Z 405.733,A -85,B 0,C 180,E1 -27184.255,E2 -27184.255} C_VEL
LIN {X 0,Y 145.758,Z 417.16,A -85,B 0,C 180,E1 -27186.025,E2 -27186.025} C_VEL
LIN {X 0,Y 138.653,Z 427.22,A -85,B 0,C 180,E1 -27188.158,E2 -27188.158} C_VEL
LIN {X 0,Y 130.617,Z 436.605,A -85,B 0,C 180,E1 -27190.899,E2 -27190.899} C_VEL
LIN {X 0,Y 123.103,Z 444.082,A -85,B 0,C 180,E1 -27193.942,E2 -27193.942} C_VEL
LIN {X 0,Y 115.253,Z 450.753,A -85,B 0,C 180,E1 -27197.752,E2 -27197.752} C_VEL
LIN {X 0,Y 106.821,Z 456.753,A -85,B 0,C 180,E1 -27202.914,E2 -27202.914} C_VEL
LIN {X 0,Y 99.933,Z 460.839,A -85,B 0,C 180,E1 -27208.396,E2 -27208.396} C_VEL
LIN {X 0,Y 94.018,Z 463.695,A -85,B 0,C 180,E1 -27214.686,E2 -27214.686} C_VEL
LIN {X 0,Y 90.792,Z 464.936,A -85,B 0,C 180,E1 -27219.278,E2 -27219.278} C_VEL
LIN {X 0,Y 86.958,Z 465.828,A -85,B 0,C 180,E1 -27226.668,E2 -27226.668} C_VEL
LIN {X 0,Y 83.995,Z 465.348,A -85,B 0,C 180,E1 -27236.796,E2 -27236.796} C_VEL
LIN {X 0,Y 83.26,Z 463.664,A -85,B 0,C 180,E1 -27245.035,E2 -27245.035} C_VEL
LIN {X 0,Y 83.919,Z 460.905,A -85,B 0,C 180,E1 -27252.955,E2 -27252.955} C_VEL
LIN {X 0,Y 85.675,Z 457.015,A -85,B 0,C 180,E1 -27260.557,E2 -27260.557} C_VEL
LIN {X 0,Y 88.335,Z 451.928,A -85,B 0,C 180,E1 -27267.719,E2 -27267.719} C_VEL
LIN {X 0,Y 92.073,Z 445.471,A -85,B 0,C 180,E1 -27274.377,E2 -27274.377} C_VEL
LIN {X 0,Y 96.831,Z 437.376,A -85,B 0,C 180,E1 -27280.453,E2 -27280.453} C_VEL
LIN {X 0,Y 102.189,Z 427.686,A -85,B 0,C 180,E1 -27285.667,E2 -27285.667} C_VEL
LIN {X 0,Y 107.157,Z 417.663,A -85,B 0,C 180,E1 -27289.64,E2 -27289.64} C_VEL
LIN {X 0,Y 111.7,Z 407.244,A -85,B 0,C 180,E1 -27292.666,E2 -27292.666} C_VEL
LIN {X 0,Y 115.829,Z 395.9,A -85,B 0,C 180,E1 -27295.133,E2 -27295.133} C_VEL
LIN {X 0,Y 119.327,Z 384.089,A -85,B 0,C 180,E1 -27297.001,E2 -27297.001} C_VEL
LIN {X 0,Y 121.992,Z 371.591,A -85,B 0,C 180,E1 -27298.437,E2 -27298.437} C_VEL
LIN {X 0,Y 124.025,Z 357.739,A -85,B 0,C 180,E1 -27299.376,E2 -27299.376} C_VEL
LIN {X 0,Y 126.736,Z 329.195,A -85,B 0,C 180,E1 -27300.628,E2 -27300.628} C_VEL
LIN {X 0,Y 125.705,Z 326.316,A -85,B 0,C 180,E1 -27301.39,E2 -27301.39} C_VEL
LIN {X 0,Y 121.186,Z 316.824,A -85,B 0,C 180,E1 -27304.724,E2 -27304.724} C_VEL
LIN {X 0,Y 116.681,Z 308.452,A -85,B 0,C 180,E1 -27308.461,E2 -27308.461} C_VEL
LIN {X 0,Y 112.111,Z 300.976,A -85,B 0,C 180,E1 -27312.759,E2 -27312.759} C_VEL
LIN {X 0,Y 107.95,Z 294.803,A -85,B 0,C 180,E1 -27317.439,E2 -27317.439} C_VEL
LIN {X 0,Y 105.288,Z 290.979,A -85,B 0,C 180,E1 -27320.984,E2 -27320.984} C_VEL
LIN {X 0,Y 102.759,Z 287.874,A -85,B 0,C 180,E1 -27324.974,E2 -27324.974} C_VEL
LIN {X 0,Y 101.971,Z 286.253,A -85,B 0,C 180,E1 -27326.538,E2 -27326.538} C_VEL
LIN {X 0,Y 98.956,Z 283.286,A -85,B 0,C 180,E1 -27333.292,E2 -27333.292} C_VEL
LIN {X 0,Y 98.138,Z 280.943,A -85,B 0,C 180,E1 -27336.569,E2 -27336.569} C_VEL
LIN {X 0,Y 96.667,Z 280.028,A -85,B 0,C 180,E1 -27347.402,E2 -27347.402} C_VEL
LIN {X 0,Y 98.659,Z 280.636,A -85,B 0,C 180,E1 -27359.531,E2 -27359.531} C_VEL
LIN {X 0,Y 99.749,Z 283.618,A -85,B 0,C 180,E1 -27363.281,E2 -27363.281} C_VEL
LIN {X 0,Y 102.424,Z 286.415,A -85,B 0,C 180,E1 -27368.819,E2 -27368.819} C_VEL
LIN {X 0,Y 104.373,Z 289.759,A -85,B 0,C 180,E1 -27372.257,E2 -27372.257} C_VEL
LIN {X 0,Y 105.888,Z 291.527,A -85,B 0,C 180,E1 -27374.417,E2 -27374.417} C_VEL
LIN {X 0,Y 109.163,Z 296.365,A -85,B 0,C 180,E1 -27378.595,E2 -27378.595} C_VEL
LIN {X 0,Y 111.817,Z 300.503,A -85,B 0,C 180,E1 -27381.542,E2 -27381.542} C_VEL
LIN {X 0,Y 115.371,Z 306.182,A -85,B 0,C 180,E1 -27384.971,E2 -27384.971} C_VEL
LIN {X 0,Y 119.804,Z 314.381,A -85,B 0,C 180,E1 -27388.808,E2 -27388.808} C_VEL
LIN {X 0,Y 123.928,Z 325.604,A -85,B 0,C 180,E1 -27392.237,E2 -27392.237} C_VEL
LIN {X 0,Y 126.463,Z 333.717,A -85,B 0,C 180,E1 -27394.247,E2 -27394.247} C_VEL
LIN {X 0,Y 123.188,Z 368.137,A -85,B 0,C 180,E1 -27395.9,E2 -27395.9} C_VEL
LIN {X 0,Y 120.647,Z 381.565,A -85,B 0,C 180,E1 -27396.952,E2 -27396.952} C_VEL
LIN {X 0,Y 117.731,Z 393.183,A -85,B 0,C 180,E1 -27398.419,E2 -27398.419} C_VEL
LIN {X 0,Y 114.01,Z 404.228,A -85,B 0,C 180,E1 -27400.286,E2 -27400.286} C_VEL
LIN {X 0,Y 109.969,Z 414.533,A -85,B 0,C 180,E1 -27402.698,E2 -27402.698} C_VEL
LIN {X 0,Y 105.028,Z 425.206,A -85,B 0,C 180,E1 -27406.034,E2 -27406.034} C_VEL
LIN {X 0,Y 100.518,Z 433.938,A -85,B 0,C 180,E1 -27409.705,E2 -27409.705} C_VEL
LIN {X 0,Y 96.02,Z 441.97,A -85,B 0,C 180,E1 -27414.16,E2 -27414.16} C_VEL
LIN {X 0,Y 91.558,Z 449.824,A -85,B 0,C 180,E1 -27420.071,E2 -27420.071} C_VEL
LIN {X 0,Y 87.916,Z 456.069,A -85,B 0,C 180,E1 -27426.442,E2 -27426.442} C_VEL
LIN {X 0,Y 85.503,Z 461.024,A -85,B 0,C 180,E1 -27433.281,E2 -27433.281} C_VEL
LIN {X 0,Y 84.201,Z 464.815,A -85,B 0,C 180,E1 -27440.391,E2 -27440.391} C_VEL
LIN {X 0,Y 83.864,Z 466.75,A -85,B 0,C 180,E1 -27445.194,E2 -27445.194} C_VEL
LIN {X 0,Y 83.915,Z 468.254,A -85,B 0,C 180,E1 -27450.001,E2 -27450.001} C_VEL
LIN {X 0,Y 83.862,Z 469.274,A -85,B 0,C 180,E1 -27454.808,E2 -27454.808} C_VEL
LIN {X 0,Y 84.971,Z 470.148,A -85,B 0,C 180,E1 -27464.368,E2 -27464.368} C_VEL
LIN {X 0,Y 88.111,Z 469.518,A -85,B 0,C 180,E1 -27473.505,E2 -27473.505} C_VEL
LIN {X 0,Y 93.472,Z 467.31,A -85,B 0,C 180,E1 -27481.758,E2 -27481.758} C_VEL
LIN {X 0,Y 98.604,Z 464.628,A -85,B 0,C 180,E1 -27487.29,E2 -27487.29} C_VEL
LIN {X 0,Y 105.548,Z 460.347,A -85,B 0,C 180,E1 -27492.909,E2 -27492.909} C_VEL
LIN {X 0,Y 113.561,Z 454.494,A -85,B 0,C 180,E1 -27497.958,E2 -27497.958} C_VEL
LIN {X 0,Y 121.098,Z 448.158,A -85,B 0,C 180,E1 -27501.581,E2 -27501.581} C_VEL
LIN {X 0,Y 129.079,Z 440.303,A -85,B 0,C 180,E1 -27504.757,E2 -27504.757} C_VEL
LIN {X 0,Y 135.934,Z 432.38,A -85,B 0,C 180,E1 -27507.156,E2 -27507.156} C_VEL
LIN {X 0,Y 143.946,Z 421.696,A -85,B 0,C 180,E1 -27509.375,E2 -27509.375} C_VEL
LIN {X 0,Y 150.574,Z 410.757,A -85,B 0,C 180,E1 -27511.063,E2 -27511.063} C_VEL
LIN {X 0,Y 156.613,Z 398.426,A -85,B 0,C 180,E1 -27512.41,E2 -27512.41} C_VEL
LIN {X 0,Y 161.403,Z 385.728,A -85,B 0,C 180,E1 -27513.37,E2 -27513.37} C_VEL
LIN {X 0,Y 165.106,Z 371.947,A -85,B 0,C 180,E1 -27514.064,E2 -27514.064} C_VEL
LIN {X 0,Y 167.207,Z 359.41,A -85,B 0,C 180,E1 -27514.499,E2 -27514.499} C_VEL
LIN {X 0,Y 167.204,Z 358.592,A -85,B 0,C 180,E1 -27514.647,E2 -27514.647} C_VEL
LIN {X 0,Y 166.076,Z 354.413,A -85,B 0,C 180,E1 -27517.038,E2 -27517.038} C_VEL
LIN {X 0,Y 165.353,Z 351.755,A -85,B 0,C 180,E1 -27518.988,E2 -27518.988} C_VEL
LIN {X 0,Y 165.055,Z 351.1,A -85,B 0,C 180,E1 -27519.789,E2 -27519.789} C_VEL
LIN {X 0,Y 164.275,Z 350.823,A -85,B 0,C 180,E1 -27521.833,E2 -27521.833} C_VEL
LIN {X 0,Y 163.277,Z 352.157,A -85,B 0,C 180,E1 -27525.262,E2 -27525.262} C_VEL
LIN {X 0,Y 162.886,Z 354.395,A -85,B 0,C 180,E1 -27529.427,E2 -27529.427} C_VEL
LIN {X 0,Y 163.027,Z 354.763,A -85,B 0,C 180,E1 -27530.832,E2 -27530.832} C_VEL
LIN {X 0,Y 163.311,Z 355.221,A -85,B 0,C 180,E1 -27532.432,E2 -27532.432} C_VEL
LIN {X 0,Y 164.146,Z 358.011,A -85,B 0,C 180,E1 -27535.753,E2 -27535.753} C_VEL
LIN {X 0,Y 165.133,Z 361.31,A -85,B 0,C 180,E1 -27538.562,E2 -27538.562} C_VEL
LIN {X 0,Y 162.682,Z 373.589,A -85,B 0,C 180,E1 -27539.024,E2 -27539.024} C_VEL
LIN {X 0,Y 158.785,Z 386.551,A -85,B 0,C 180,E1 -27539.818,E2 -27539.818} C_VEL
LIN {X 0,Y 153.755,Z 398.918,A -85,B 0,C 180,E1 -27540.877,E2 -27540.877} C_VEL
LIN {X 0,Y 147.706,Z 410.509,A -85,B 0,C 180,E1 -27542.287,E2 -27542.287} C_VEL
LIN {X 0,Y 140.904,Z 420.987,A -85,B 0,C 180,E1 -27544.006,E2 -27544.006} C_VEL
LIN {X 0,Y 133.022,Z 431.029,A -85,B 0,C 180,E1 -27546.255,E2 -27546.255} C_VEL
LIN {X 0,Y 124.687,Z 439.807,A -85,B 0,C 180,E1 -27549.045,E2 -27549.045} C_VEL
LIN {X 0,Y 116.827,Z 446.796,A -85,B 0,C 180,E1 -27552.161,E2 -27552.161} C_VEL
LIN {X 0,Y 109.477,Z 452.38,A -85,B 0,C 180,E1 -27555.646,E2 -27555.646} C_VEL
LIN {X 0,Y 101.742,Z 457.406,A -85,B 0,C 180,E1 -27560.206,E2 -27560.206} C_VEL
LIN {X 0,Y 93.971,Z 461.597,A -85,B 0,C 180,E1 -27566.172,E2 -27566.172} C_VEL
LIN {X 0,Y 89.66,Z 463.475,A -85,B 0,C 180,E1 -27570.43,E2 -27570.43} C_VEL
LIN {X 0,Y 85.89,Z 464.849,A -85,B 0,C 180,E1 -27575.089,E2 -27575.089} C_VEL
LIN {X 0,Y 82.676,Z 465.715,A -85,B 0,C 180,E1 -27580.087,E2 -27580.087} C_VEL
LIN {X 0,Y 80.101,Z 466.06,A -85,B 0,C 180,E1 -27585.419,E2 -27585.419} C_VEL
LIN {X 0,Y 77.184,Z 465.569,A -85,B 0,C 180,E1 -27595.036,E2 -27595.036} C_VEL
LIN {X 0,Y 76.244,Z 464.236,A -85,B 0,C 180,E1 -27602.555,E2 -27602.555} C_VEL
LIN {X 0,Y 76.556,Z 461.692,A -85,B 0,C 180,E1 -27611.257,E2 -27611.257} C_VEL
LIN {X 0,Y 78.404,Z 457.631,A -85,B 0,C 180,E1 -27620.412,E2 -27620.412} C_VEL
LIN {X 0,Y 80.829,Z 453.193,A -85,B 0,C 180,E1 -27627.508,E2 -27627.508} C_VEL
LIN {X 0,Y 84.649,Z 446.979,A -85,B 0,C 180,E1 -27634.762,E2 -27634.762} C_VEL
LIN {X 0,Y 89.511,Z 439.193,A -85,B 0,C 180,E1 -27641.319,E2 -27641.319} C_VEL
LIN {X 0,Y 94.323,Z 431.21,A -85,B 0,C 180,E1 -27646.224,E2 -27646.224} C_VEL
LIN {X 0,Y 99.625,Z 421.471,A -85,B 0,C 180,E1 -27650.653,E2 -27650.653} C_VEL
LIN {X 0,Y 104.898,Z 410.529,A -85,B 0,C 180,E1 -27654.227,E2 -27654.227} C_VEL
LIN {X 0,Y 109.584,Z 398.978,A -85,B 0,C 180,E1 -27656.992,E2 -27656.992} C_VEL
LIN {X 0,Y 113.537,Z 386.78,A -85,B 0,C 180,E1 -27659.075,E2 -27659.075} C_VEL
LIN {X 0,Y 116.742,Z 373.283,A -85,B 0,C 180,E1 -27660.721,E2 -27660.721} C_VEL
LIN {X 0,Y 118.862,Z 360.397,A -85,B 0,C 180,E1 -27661.676,E2 -27661.676} C_VEL
LIN {X 0,Y 121.722,Z 331.029,A -85,B 0,C 180,E1 -27663.027,E2 -27663.027} C_VEL
LIN {X 0,Y 117.655,Z 322.007,A -85,B 0,C 180,E1 -27666.334,E2 -27666.334} C_VEL
LIN {X 0,Y 113.339,Z 313.659,A -85,B 0,C 180,E1 -27670.216,E2 -27670.216} C_VEL
LIN {X 0,Y 108.662,Z 305.504,A -85,B 0,C 180,E1 -27675.167,E2 -27675.167} C_VEL
LIN {X 0,Y 105.288,Z 300.524,A -85,B 0,C 180,E1 -27679.346,E2 -27679.346} C_VEL
LIN {X 0,Y 103.151,Z 297.271,A -85,B 0,C 180,E1 -27682.517,E2 -27682.517} C_VEL
LIN {X 0,Y 100.786,Z 293.973,A -85,B 0,C 180,E1 -27686.692,E2 -27686.692} C_VEL
LIN {X 0,Y 99.997,Z 292.706,A -85,B 0,C 180,E1 -27688.336,E2 -27688.336} C_VEL
LIN {X 0,Y 97.541,Z 289.812,A -85,B 0,C 180,E1 -27694.708,E2 -27694.708} C_VEL
LIN {X 0,Y 96.852,Z 287.76,A -85,B 0,C 180,E1 -27697.858,E2 -27697.858} C_VEL
LIN {X 0,Y 95.727,Z 287.08,A -85,B 0,C 180,E1 -27707.276,E2 -27707.276} C_VEL
LIN {X 0,Y 97.227,Z 287.52,A -85,B 0,C 180,E1 -27717.966,E2 -27717.966} C_VEL
LIN {X 0,Y 97.548,Z 288.298,A -85,B 0,C 180,E1 -27719.324,E2 -27719.324} C_VEL
LIN {X 0,Y 98.946,Z 291.203,A -85,B 0,C 180,E1 -27723.818,E2 -27723.818} C_VEL
LIN {X 0,Y 100.691,Z 293.012,A -85,B 0,C 180,E1 -27727.52,E2 -27727.52} C_VEL
LIN {X 0,Y 102.786,Z 296.554,A -85,B 0,C 180,E1 -27731.462,E2 -27731.462} C_VEL
LIN {X 0,Y 103.978,Z 298.203,A -85,B 0,C 180,E1 -27733.315,E2 -27733.315} C_VEL
LIN {X 0,Y 106.835,Z 302.607,A -85,B 0,C 180,E1 -27737.223,E2 -27737.223} C_VEL
LIN {X 0,Y 109.538,Z 307.023,A -85,B 0,C 180,E1 -27740.456,E2 -27740.456} C_VEL
LIN {X 0,Y 113.704,Z 314.38,A -85,B 0,C 180,E1 -27744.735,E2 -27744.735} C_VEL
LIN {X 0,Y 116.348,Z 319.766,A -85,B 0,C 180,E1 -27747.182,E2 -27747.182} C_VEL
LIN {X 0,Y 120.237,Z 331.145,A -85,B 0,C 180,E1 -27750.76,E2 -27750.76} C_VEL
LIN {X 0,Y 121.515,Z 335.66,A -85,B 0,C 180,E1 -27751.907,E2 -27751.907} C_VEL
LIN {X 0,Y 118.305,Z 367.873,A -85,B 0,C 180,E1 -27753.461,E2 -27753.461} C_VEL
LIN {X 0,Y 115.666,Z 381.338,A -85,B 0,C 180,E1 -27754.507,E2 -27754.507} C_VEL
LIN {X 0,Y 112.459,Z 393.476,A -85,B 0,C 180,E1 -27756.05,E2 -27756.05} C_VEL
LIN {X 0,Y 108.29,Z 405.201,A -85,B 0,C 180,E1 -27758.104,E2 -27758.104} C_VEL
LIN {X 0,Y 103.473,Z 416.587,A -85,B 0,C 180,E1 -27760.922,E2 -27760.922} C_VEL
LIN {X 0,Y 98.388,Z 426.861,A -85,B 0,C 180,E1 -27764.414,E2 -27764.414} C_VEL
LIN {X 0,Y 93.096,Z 436.225,A -85,B 0,C 180,E1 -27768.782,E2 -27768.782} C_VEL
LIN {X 0,Y 88.668,Z 443.717,A -85,B 0,C 180,E1 -27773.527,E2 -27773.527} C_VEL
LIN {X 0,Y 84.005,Z 451.168,A -85,B 0,C 180,E1 -27779.871,E2 -27779.871} C_VEL
LIN {X 0,Y 80.379,Z 457.122,A -85,B 0,C 180,E1 -27786.831,E2 -27786.831} C_VEL
LIN {X 0,Y 78.094,Z 461.81,A -85,B 0,C 180,E1 -27794.338,E2 -27794.338} C_VEL
LIN {X 0,Y 77.203,Z 464.278,A -85,B 0,C 180,E1 -27799.511,E2 -27799.511} C_VEL
LIN {X 0,Y 76.784,Z 466.268,A -85,B 0,C 180,E1 -27804.749,E2 -27804.749} C_VEL
LIN {X 0,Y 76.833,Z 467.831,A -85,B 0,C 180,E1 -27810.001,E2 -27810.001} C_VEL
LIN {X 0,Y 76.782,Z 468.945,A -85,B 0,C 180,E1 -27815.253,E2 -27815.253} C_VEL
LIN {X 0,Y 77.187,Z 469.625,A -85,B 0,C 180,E1 -27820.493,E2 -27820.493} C_VEL
LIN {X 0,Y 79.596,Z 469.854,A -85,B 0,C 180,E1 -27830.683,E2 -27830.683} C_VEL
LIN {X 0,Y 81.62,Z 469.416,A -85,B 0,C 180,E1 -27835.502,E2 -27835.502} C_VEL
LIN {X 0,Y 84.32,Z 468.593,A -85,B 0,C 180,E1 -27840.007,E2 -27840.007} C_VEL
LIN {X 0,Y 91.076,Z 465.743,A -85,B 0,C 180,E1 -27848.122,E2 -27848.122} C_VEL
LIN {X 0,Y 97.275,Z 462.538,A -85,B 0,C 180,E1 -27853.344,E2 -27853.344} C_VEL
LIN {X 0,Y 104.054,Z 458.331,A -85,B 0,C 180,E1 -27857.985,E2 -27857.985} C_VEL
LIN {X 0,Y 112.809,Z 452.005,A -85,B 0,C 180,E1 -27862.592,E2 -27862.592} C_VEL
LIN {X 0,Y 120.945,Z 445.172,A -85,B 0,C 180,E1 -27865.9,E2 -27865.9} C_VEL
LIN {X 0,Y 129.38,Z 436.706,A -85,B 0,C 180,E1 -27868.821,E2 -27868.821} C_VEL
LIN {X 0,Y 136.76,Z 428.058,A -85,B 0,C 180,E1 -27870.882,E2 -27870.882} C_VEL
LIN {X 0,Y 144.294,Z 417.49,A -85,B 0,C 180,E1 -27872.734,E2 -27872.734} C_VEL
LIN {X 0,Y 150.412,Z 407.035,A -85,B 0,C 180,E1 -27874.087,E2 -27874.087} C_VEL
LIN {X 0,Y 156.071,Z 394.917,A -85,B 0,C 180,E1 -27875.2,E2 -27875.2} C_VEL
LIN {X 0,Y 160.726,Z 381.899,A -85,B 0,C 180,E1 -27876.019,E2 -27876.019} C_VEL
LIN {X 0,Y 163.919,Z 369.117,A -85,B 0,C 180,E1 -27876.558,E2 -27876.558} C_VEL
LIN {X 0,Y 165.005,Z 362.661,A -85,B 0,C 180,E1 -27876.811,E2 -27876.811} C_VEL
LIN {X 0,Y 164.105,Z 358.454,A -85,B 0,C 180,E1 -27879.681,E2 -27879.681} C_VEL
LIN {X 0,Y 163.009,Z 354.916,A -85,B 0,C 180,E1 -27884.608,E2 -27884.608} C_VEL
LIN {X 0,Y 163.027,Z 354.763,A -85,B 0,C 180,E1 -27890.832,E2 -27890.832} C_VEL
LIN {X 0,Y 163.23,Z 355.681,A -85,B 0,C 180,E1 -27892.284,E2 -27892.284} C_VEL
LIN {X 0,Y 163.353,Z 357.708,A -85,B 0,C 180,E1 -27893.606,E2 -27893.606} C_VEL
LIN {X 0,Y 163.347,Z 360.513,A -85,B 0,C 180,E1 -27894.749,E2 -27894.749} C_VEL
LIN {X 0,Y 163.141,Z 363.919,A -85,B 0,C 180,E1 -27895.664,E2 -27895.664} C_VEL
LIN {X 0,Y 162.618,Z 367.78,A -85,B 0,C 180,E1 -27896.26,E2 -27896.26} C_VEL
LIN {X 0,Y 162.347,Z 369.14,A -85,B 0,C 180,E1 -27896.364,E2 -27896.364} C_VEL
LIN {X 0,Y 159.087,Z 381.392,A -85,B 0,C 180,E1 -27896.966,E2 -27896.966} C_VEL
LIN {X 0,Y 154.284,Z 394.321,A -85,B 0,C 180,E1 -27897.864,E2 -27897.864} C_VEL
LIN {X 0,Y 148.487,Z 406.145,A -85,B 0,C 180,E1 -27899.038,E2 -27899.038} C_VEL
LIN {X 0,Y 141.596,Z 417.285,A -85,B 0,C 180,E1 -27900.536,E2 -27900.536} C_VEL
LIN {X 0,Y 133.661,Z 427.779,A -85,B 0,C 180,E1 -27902.515,E2 -27902.515} C_VEL
LIN {X 0,Y 125.21,Z 436.933,A -85,B 0,C 180,E1 -27904.927,E2 -27904.927} C_VEL
LIN {X 0,Y 117.009,Z 444.385,A -85,B 0,C 180,E1 -27907.67,E2 -27907.67} C_VEL
LIN {X 0,Y 107.585,Z 451.556,A -85,B 0,C 180,E1 -27911.514,E2 -27911.514} C_VEL
LIN {X 0,Y 97.781,Z 457.603,A -85,B 0,C 180,E1 -27916.709,E2 -27916.709} C_VEL
LIN {X 0,Y 90.705,Z 461.178,A -85,B 0,C 180,E1 -27921.599,E2 -27921.599} C_VEL
LIN {X 0,Y 85.839,Z 463.241,A -85,B 0,C 180,E1 -27925.761,E2 -27925.761} C_VEL
LIN {X 0,Y 80.565,Z 465.007,A -85,B 0,C 180,E1 -27931.561,E2 -27931.561} C_VEL
LIN {X 0,Y 74.588,Z 466.232,A -85,B 0,C 180,E1 -27941.079,E2 -27941.079} C_VEL
LIN {X 0,Y 72.107,Z 466.222,A -85,B 0,C 180,E1 -27946.978,E2 -27946.978} C_VEL
LIN {X 0,Y 70.384,Z 465.76,A -85,B 0,C 180,E1 -27953.193,E2 -27953.193} C_VEL
LIN {X 0,Y 69.339,Z 464.79,A -85,B 0,C 180,E1 -27959.549,E2 -27959.549} C_VEL
LIN {X 0,Y 69.077,Z 463.264,A -85,B 0,C 180,E1 -27966.303,E2 -27966.303} C_VEL
LIN {X 0,Y 70.045,Z 460.264,A -85,B 0,C 180,E1 -27975.472,E2 -27975.472} C_VEL
LIN {X 0,Y 72.315,Z 456.048,A -85,B 0,C 180,E1 -27984.422,E2 -27984.422} C_VEL
LIN {X 0,Y 75.79,Z 450.582,A -85,B 0,C 180,E1 -27992.657,E2 -27992.657} C_VEL
LIN {X 0,Y 80.412,Z 443.644,A -85,B 0,C 180,E1 -28000.066,E2 -28000.066} C_VEL
LIN {X 0,Y 86.152,Z 434.976,A -85,B 0,C 180,E1 -28006.589,E2 -28006.589} C_VEL
LIN {X 0,Y 91.863,Z 425.571,A -85,B 0,C 180,E1 -28011.569,E2 -28011.569} C_VEL
LIN {X 0,Y 97.552,Z 414.917,A -85,B 0,C 180,E1 -28015.61,E2 -28015.61} C_VEL
LIN {X 0,Y 102.668,Z 403.803,A -85,B 0,C 180,E1 -28018.631,E2 -28018.631} C_VEL
LIN {X 0,Y 107.355,Z 391.071,A -85,B 0,C 180,E1 -28021.098,E2 -28021.098} C_VEL
LIN {X 0,Y 110.968,Z 378.197,A -85,B 0,C 180,E1 -28022.866,E2 -28022.866} C_VEL
LIN {X 0,Y 113.436,Z 365.685,A -85,B 0,C 180,E1 -28023.995,E2 -28023.995} C_VEL
LIN {X 0,Y 115.613,Z 347.431,A -85,B 0,C 180,E1 -28024.907,E2 -28024.907} C_VEL
LIN {X 0,Y 116.957,Z 333.518,A -85,B 0,C 180,E1 -28025.547,E2 -28025.547} C_VEL
LIN {X 0,Y 113.16,Z 324.946,A -85,B 0,C 180,E1 -28029.011,E2 -28029.011} C_VEL
LIN {X 0,Y 109.402,Z 317.431,A -85,B 0,C 180,E1 -28032.855,E2 -28032.855} C_VEL
LIN {X 0,Y 105.877,Z 311.148,A -85,B 0,C 180,E1 -28037.026,E2 -28037.026} C_VEL
LIN {X 0,Y 102.951,Z 306.501,A -85,B 0,C 180,E1 -28041.049,E2 -28041.049} C_VEL
LIN {X 0,Y 101.228,Z 303.709,A -85,B 0,C 180,E1 -28043.885,E2 -28043.885} C_VEL
LIN {X 0,Y 98.95,Z 300.196,A -85,B 0,C 180,E1 -28048.322,E2 -28048.322} C_VEL
LIN {X 0,Y 98.23,Z 299.252,A -85,B 0,C 180,E1 -28049.945,E2 -28049.945} C_VEL
LIN {X 0,Y 96.073,Z 296.071,A -85,B 0,C 180,E1 -28056.624,E2 -28056.624} C_VEL
LIN {X 0,Y 95.736,Z 294.828,A -85,B 0,C 180,E1 -28058.466,E2 -28058.466} C_VEL
LIN {X 0,Y 94.789,Z 294.122,A -85,B 0,C 180,E1 -28067.148,E2 -28067.148} C_VEL
LIN {X 0,Y 96.083,Z 294.512,A -85,B 0,C 180,E1 -28077.256,E2 -28077.256} C_VEL
LIN {X 0,Y 97.644,Z 298.069,A -85,B 0,C 180,E1 -28083.058,E2 -28083.058} C_VEL
LIN {X 0,Y 99.064,Z 299.755,A -85,B 0,C 180,E1 -28086.363,E2 -28086.363} C_VEL
LIN {X 0,Y 101.343,Z 303.511,A -85,B 0,C 180,E1 -28090.852,E2 -28090.852} C_VEL
LIN {X 0,Y 104.55,Z 308.855,A -85,B 0,C 180,E1 -28095.813,E2 -28095.813} C_VEL
LIN {X 0,Y 107.83,Z 314.484,A -85,B 0,C 180,E1 -28099.956,E2 -28099.956} C_VEL
LIN {X 0,Y 112.306,Z 323.316,A -85,B 0,C 180,E1 -28104.778,E2 -28104.778} C_VEL
LIN {X 0,Y 115.443,Z 332.853,A -85,B 0,C 180,E1 -28108.028,E2 -28108.028} C_VEL
LIN {X 0,Y 116.795,Z 337.561,A -85,B 0,C 180,E1 -28109.387,E2 -28109.387} C_VEL
LIN {X 0,Y 113.645,Z 367.499,A -85,B 0,C 180,E1 -28110.806,E2 -28110.806} C_VEL
LIN {X 0,Y 110.973,Z 380.871,A -85,B 0,C 180,E1 -28111.836,E2 -28111.836} C_VEL
LIN {X 0,Y 107.732,Z 392.71,A -85,B 0,C 180,E1 -28113.299,E2 -28113.299} C_VEL
LIN {X 0,Y 103.371,Z 404.565,A -85,B 0,C 180,E1 -28115.329,E2 -28115.329} C_VEL
LIN {X 0,Y 98.965,Z 414.748,A -85,B 0,C 180,E1 -28117.812,E2 -28117.812} C_VEL
LIN {X 0,Y 93.509,Z 425.311,A -85,B 0,C 180,E1 -28121.274,E2 -28121.274} C_VEL
LIN {X 0,Y 87.925,Z 434.838,A -85,B 0,C 180,E1 -28125.624,E2 -28125.624} C_VEL
LIN {X 0,Y 82.975,Z 442.638,A -85,B 0,C 180,E1 -28130.563,E2 -28130.563} C_VEL
LIN {X 0,Y 77.919,Z 450.255,A -85,B 0,C 180,E1 -28137.237,E2 -28137.237} C_VEL
LIN {X 0,Y 73.861,Z 456.342,A -85,B 0,C 180,E1 -28144.649,E2 -28144.649} C_VEL
LIN {X 0,Y 71.244,Z 461.155,A -85,B 0,C 180,E1 -28152.787,E2 -28152.787} C_VEL
LIN {X 0,Y 69.889,Z 464.805,A -85,B 0,C 180,E1 -28161.325,E2 -28161.325} C_VEL
LIN {X 0,Y 69.737,Z 467.402,A -85,B 0,C 180,E1 -28170.001,E2 -28170.001} C_VEL
LIN {X 0,Y 69.725,Z 468.574,A -85,B 0,C 180,E1 -28175.786,E2 -28175.786} C_VEL
LIN {X 0,Y 70.197,Z 469.344,A -85,B 0,C 180,E1 -28181.552,E2 -28181.552} C_VEL
LIN {X 0,Y 72.965,Z 469.683,A -85,B 0,C 180,E1 -28192.662,E2 -28192.662} C_VEL
LIN {X 0,Y 78.23,Z 468.553,A -85,B 0,C 180,E1 -28202.618,E2 -28202.618} C_VEL
LIN {X 0,Y 81.721,Z 467.412,A -85,B 0,C 180,E1 -28207.014,E2 -28207.014} C_VEL
LIN {X 0,Y 85.596,Z 465.852,A -85,B 0,C 180,E1 -28211.061,E2 -28211.061} C_VEL
LIN {X 0,Y 93.002,Z 462.36,A -85,B 0,C 180,E1 -28216.927,E2 -28216.927} C_VEL
LIN {X 0,Y 102,Z 457.113,A -85,B 0,C 180,E1 -28222.408,E2 -28222.408} C_VEL
LIN {X 0,Y 111.455,Z 450.492,A -85,B 0,C 180,E1 -28226.668,E2 -28226.668} C_VEL
LIN {X 0,Y 120.076,Z 443.313,A -85,B 0,C 180,E1 -28229.691,E2 -28229.691} C_VEL
LIN {X 0,Y 127.352,Z 436.105,A -85,B 0,C 180,E1 -28232.003,E2 -28232.003} C_VEL
LIN {X 0,Y 135.03,Z 427.36,A -85,B 0,C 180,E1 -28233.873,E2 -28233.873} C_VEL
LIN {X 0,Y 142.787,Z 416.721,A -85,B 0,C 180,E1 -28235.585,E2 -28235.585} C_VEL
LIN {X 0,Y 149.089,Z 406.118,A -85,B 0,C 180,E1 -28236.813,E2 -28236.813} C_VEL
LIN {X 0,Y 154.626,Z 394.474,A -85,B 0,C 180,E1 -28237.789,E2 -28237.789} C_VEL
LIN {X 0,Y 159.216,Z 381.947,A -85,B 0,C 180,E1 -28238.504,E2 -28238.504} C_VEL
LIN {X 0,Y 162.523,Z 369.154,A -85,B 0,C 180,E1 -28239,E2 -28239} C_VEL
LIN {X 0,Y 162.92,Z 366.862,A -85,B 0,C 180,E1 -28239.152,E2 -28239.152} C_VEL
LIN {X 0,Y 162.642,Z 364.872,A -85,B 0,C 180,E1 -28240.658,E2 -28240.658} C_VEL
LIN {X 0,Y 161.934,Z 361.966,A -85,B 0,C 180,E1 -28244.906,E2 -28244.906} C_VEL
LIN {X 0,Y 161.983,Z 361.777,A -85,B 0,C 180,E1 -28250.743,E2 -28250.743} C_VEL
LIN {X 0,Y 162.177,Z 362.254,A -85,B 0,C 180,E1 -28252.075,E2 -28252.075} C_VEL
LIN {X 0,Y 162.721,Z 364.785,A -85,B 0,C 180,E1 -28255.157,E2 -28255.157} C_VEL
LIN {X 0,Y 162.976,Z 365.875,A -85,B 0,C 180,E1 -28256.213,E2 -28256.213} C_VEL
LIN {X 0,Y 162.347,Z 369.14,A -85,B 0,C 180,E1 -28256.364,E2 -28256.364} C_VEL
LIN {X 0,Y 161.407,Z 373.013,A -85,B 0,C 180,E1 -28256.447,E2 -28256.447} C_VEL
LIN {X 0,Y 159.011,Z 380.449,A -85,B 0,C 180,E1 -28256.11,E2 -28256.11} C_VEL
LIN {X 0,Y 156.108,Z 387.731,A -85,B 0,C 180,E1 -28255.584,E2 -28255.584} C_VEL
LIN {X 0,Y 152.86,Z 394.974,A -85,B 0,C 180,E1 -28255.379,E2 -28255.379} C_VEL
LIN {X 0,Y 151.192,Z 398.435,A -85,B 0,C 180,E1 -28255.549,E2 -28255.549} C_VEL
LIN {X 0,Y 144.803,Z 410.244,A -85,B 0,C 180,E1 -28256.759,E2 -28256.759} C_VEL
LIN {X 0,Y 137.999,Z 420.276,A -85,B 0,C 180,E1 -28258.117,E2 -28258.117} C_VEL
LIN {X 0,Y 129.804,Z 430.235,A -85,B 0,C 180,E1 -28260,E2 -28260} C_VEL
LIN {X 0,Y 121.326,Z 438.779,A -85,B 0,C 180,E1 -28262.239,E2 -28262.239} C_VEL
LIN {X 0,Y 112.856,Z 445.913,A -85,B 0,C 180,E1 -28264.872,E2 -28264.872} C_VEL
LIN {X 0,Y 105.252,Z 451.331,A -85,B 0,C 180,E1 -28267.675,E2 -28267.675} C_VEL
LIN {X 0,Y 96.837,Z 456.444,A -85,B 0,C 180,E1 -28271.553,E2 -28271.553} C_VEL
LIN {X 0,Y 88.037,Z 460.781,A -85,B 0,C 180,E1 -28276.67,E2 -28276.67} C_VEL
LIN {X 0,Y 82.646,Z 462.946,A -85,B 0,C 180,E1 -28280.703,E2 -28280.703} C_VEL
LIN {X 0,Y 75.392,Z 465.228,A -85,B 0,C 180,E1 -28287.782,E2 -28287.782} C_VEL
LIN {X 0,Y 68.516,Z 466.444,A -85,B 0,C 180,E1 -28297.985,E2 -28297.985} C_VEL
LIN {X 0,Y 64.178,Z 466.123,A -85,B 0,C 180,E1 -28308.924,E2 -28308.924} C_VEL
LIN {X 0,Y 62.666,Z 465.313,A -85,B 0,C 180,E1 -28315.891,E2 -28315.891} C_VEL
LIN {X 0,Y 61.982,Z 463.515,A -85,B 0,C 180,E1 -28325.11,E2 -28325.11} C_VEL
LIN {X 0,Y 63.179,Z 459.901,A -85,B 0,C 180,E1 -28337.144,E2 -28337.144} C_VEL
LIN {X 0,Y 65.817,Z 455.47,A -85,B 0,C 180,E1 -28346.939,E2 -28346.939} C_VEL
LIN {X 0,Y 69.766,Z 449.775,A -85,B 0,C 180,E1 -28355.781,E2 -28355.781} C_VEL
LIN {X 0,Y 74.965,Z 442.62,A -85,B 0,C 180,E1 -28363.554,E2 -28363.554} C_VEL
LIN {X 0,Y 80.157,Z 435.278,A -85,B 0,C 180,E1 -28369.194,E2 -28369.194} C_VEL
LIN {X 0,Y 85.956,Z 426.366,A -85,B 0,C 180,E1 -28374.129,E2 -28374.129} C_VEL
LIN {X 0,Y 91.587,Z 416.519,A -85,B 0,C 180,E1 -28378.034,E2 -28378.034} C_VEL
LIN {X 0,Y 97.478,Z 404.525,A -85,B 0,C 180,E1 -28381.398,E2 -28381.398} C_VEL
LIN {X 0,Y 102.099,Z 392.843,A -85,B 0,C 180,E1 -28383.707,E2 -28383.707} C_VEL
LIN {X 0,Y 105.892,Z 380.345,A -85,B 0,C 180,E1 -28385.483,E2 -28385.483} C_VEL
LIN {X 0,Y 108.759,Z 367.288,A -85,B 0,C 180,E1 -28386.728,E2 -28386.728} C_VEL
LIN {X 0,Y 110.727,Z 352.545,A -85,B 0,C 180,E1 -28387.513,E2 -28387.513} C_VEL
LIN {X 0,Y 112.424,Z 336.128,A -85,B 0,C 180,E1 -28388.232,E2 -28388.232} C_VEL
LIN {X 0,Y 108.288,Z 326.622,A -85,B 0,C 180,E1 -28392.571,E2 -28392.571} C_VEL
LIN {X 0,Y 104.084,Z 318.269,A -85,B 0,C 180,E1 -28397.758,E2 -28397.758} C_VEL
LIN {X 0,Y 100.688,Z 312.413,A -85,B 0,C 180,E1 -28402.871,E2 -28402.871} C_VEL
LIN {X 0,Y 99.256,Z 310.001,A -85,B 0,C 180,E1 -28405.496,E2 -28405.496} C_VEL
LIN {X 0,Y 96.955,Z 306.144,A -85,B 0,C 180,E1 -28410.594,E2 -28410.594} C_VEL
LIN {X 0,Y 94.851,Z 302.849,A -85,B 0,C 180,E1 -28417.672,E2 -28417.672} C_VEL
LIN {X 0,Y 94.583,Z 301.808,A -85,B 0,C 180,E1 -28419.353,E2 -28419.353} C_VEL
LIN {X 0,Y 93.85,Z 301.174,A -85,B 0,C 180,E1 -28427.017,E2 -28427.017} C_VEL
LIN {X 0,Y 94.331,Z 301.304,A -85,B 0,C 180,E1 -28433.583,E2 -28433.583} C_VEL
LIN {X 0,Y 94.994,Z 301.713,A -85,B 0,C 180,E1 -28436.858,E2 -28436.858} C_VEL
LIN {X 0,Y 96.377,Z 304.953,A -85,B 0,C 180,E1 -28442.329,E2 -28442.329} C_VEL
LIN {X 0,Y 97.438,Z 306.359,A -85,B 0,C 180,E1 -28445.056,E2 -28445.056} C_VEL
LIN {X 0,Y 100.08,Z 311.092,A -85,B 0,C 180,E1 -28450.606,E2 -28450.606} C_VEL
LIN {X 0,Y 102.693,Z 315.719,A -85,B 0,C 180,E1 -28454.876,E2 -28454.876} C_VEL
LIN {X 0,Y 106.248,Z 322.458,A -85,B 0,C 180,E1 -28459.63,E2 -28459.63} C_VEL
LIN {X 0,Y 109.09,Z 328.72,A -85,B 0,C 180,E1 -28462.972,E2 -28462.972} C_VEL
LIN {X 0,Y 112.237,Z 339.436,A -85,B 0,C 180,E1 -28466.616,E2 -28466.616} C_VEL
LIN {X 0,Y 109.238,Z 367.205,A -85,B 0,C 180,E1 -28467.954,E2 -28467.954} C_VEL
LIN {X 0,Y 106.466,Z 380.618,A -85,B 0,C 180,E1 -28468.958,E2 -28468.958} C_VEL
LIN {X 0,Y 102.928,Z 392.928,A -85,B 0,C 180,E1 -28470.455,E2 -28470.455} C_VEL
LIN {X 0,Y 98.067,Z 405.48,A -85,B 0,C 180,E1 -28472.643,E2 -28472.643} C_VEL
LIN {X 0,Y 92.75,Z 416.727,A -85,B 0,C 180,E1 -28475.457,E2 -28475.457} C_VEL
LIN {X 0,Y 87.745,Z 425.864,A -85,B 0,C 180,E1 -28478.655,E2 -28478.655} C_VEL
LIN {X 0,Y 81.615,Z 435.533,A -85,B 0,C 180,E1 -28483.313,E2 -28483.313} C_VEL
LIN {X 0,Y 76.591,Z 442.94,A -85,B 0,C 180,E1 -28488.335,E2 -28488.335} C_VEL
LIN {X 0,Y 71.186,Z 450.437,A -85,B 0,C 180,E1 -28495.412,E2 -28495.412} C_VEL
LIN {X 0,Y 66.311,Z 457.341,A -85,B 0,C 180,E1 -28504.917,E2 -28504.917} C_VEL
LIN {X 0,Y 63.792,Z 461.876,A -85,B 0,C 180,E1 -28514.014,E2 -28514.014} C_VEL
LIN {X 0,Y 62.653,Z 465.283,A -85,B 0,C 180,E1 -28523.561,E2 -28523.561} C_VEL
LIN {X 0,Y 62.662,Z 466.956,A -85,B 0,C 180,E1 -28530.001,E2 -28530.001} C_VEL
LIN {X 0,Y 62.668,Z 468.183,A -85,B 0,C 180,E1 -28536.44,E2 -28536.44} C_VEL
LIN {X 0,Y 64.499,Z 469.47,A -85,B 0,C 180,E1 -28549.081,E2 -28549.081} C_VEL
LIN {X 0,Y 69.025,Z 469.185,A -85,B 0,C 180,E1 -28560.604,E2 -28560.604} C_VEL
LIN {X 0,Y 76.146,Z 467.436,A -85,B 0,C 180,E1 -28570.247,E2 -28570.247} C_VEL
LIN {X 0,Y 80.376,Z 465.979,A -85,B 0,C 180,E1 -28574.389,E2 -28574.389} C_VEL
LIN {X 0,Y 89.465,Z 462.04,A -85,B 0,C 180,E1 -28581.065,E2 -28581.065} C_VEL
LIN {X 0,Y 97.84,Z 457.511,A -85,B 0,C 180,E1 -28585.697,E2 -28585.697} C_VEL
LIN {X 0,Y 106.27,Z 452.096,A -85,B 0,C 180,E1 -28589.287,E2 -28589.287} C_VEL
LIN {X 0,Y 115.155,Z 445.376,A -85,B 0,C 180,E1 -28592.245,E2 -28592.245} C_VEL
LIN {X 0,Y 124.21,Z 437.145,A -85,B 0,C 180,E1 -28594.865,E2 -28594.865} C_VEL
LIN {X 0,Y 132.097,Z 428.675,A -85,B 0,C 180,E1 -28596.6,E2 -28596.6} C_VEL
LIN {X 0,Y 140.041,Z 418.351,A -85,B 0,C 180,E1 -28598.191,E2 -28598.191} C_VEL
LIN {X 0,Y 146.471,Z 408.206,A -85,B 0,C 180,E1 -28599.334,E2 -28599.334} C_VEL
LIN {X 0,Y 152.496,Z 396.455,A -85,B 0,C 180,E1 -28600.274,E2 -28600.274} C_VEL
LIN {X 0,Y 157.518,Z 383.529,A -85,B 0,C 180,E1 -28600.967,E2 -28600.967} C_VEL
LIN {X 0,Y 160.905,Z 371.411,A -85,B 0,C 180,E1 -28601.471,E2 -28601.471} C_VEL
LIN {X 0,Y 160.533,Z 368.866,A -85,B 0,C 180,E1 -28605.497,E2 -28605.497} C_VEL
LIN {X 0,Y 160.684,Z 368.765,A -85,B 0,C 180,E1 -28611.026,E2 -28611.026} C_VEL
LIN {X 0,Y 160.895,Z 370.863,A -85,B 0,C 180,E1 -28613.94,E2 -28613.94} C_VEL
LIN {X 0,Y 157.078,Z 384.175,A -85,B 0,C 180,E1 -28614.576,E2 -28614.576} C_VEL
LIN {X 0,Y 152.484,Z 395.728,A -85,B 0,C 180,E1 -28615.342,E2 -28615.342} C_VEL
LIN {X 0,Y 151.192,Z 398.435,A -85,B 0,C 180,E1 -28615.549,E2 -28615.549} C_VEL
LIN {X 0,Y 148.468,Z 403.665,A -85,B 0,C 180,E1 -28615.766,E2 -28615.766} C_VEL
LIN {X 0,Y 143.174,Z 412.056,A -85,B 0,C 180,E1 -28615.522,E2 -28615.522} C_VEL
LIN {X 0,Y 137.264,Z 419.972,A -85,B 0,C 180,E1 -28615.372,E2 -28615.372} C_VEL
LIN {X 0,Y 133.572,Z 424.448,A -85,B 0,C 180,E1 -28615.789,E2 -28615.789} C_VEL
LIN {X 0,Y 124.855,Z 433.975,A -85,B 0,C 180,E1 -28617.619,E2 -28617.619} C_VEL
LIN {X 0,Y 115.34,Z 442.559,A -85,B 0,C 180,E1 -28620,E2 -28620} C_VEL
LIN {X 0,Y 105.561,Z 449.753,A -85,B 0,C 180,E1 -28622.959,E2 -28622.959} C_VEL
LIN {X 0,Y 95.552,Z 455.757,A -85,B 0,C 180,E1 -28626.808,E2 -28626.808} C_VEL
LIN {X 0,Y 86.068,Z 460.327,A -85,B 0,C 180,E1 -28631.512,E2 -28631.512} C_VEL
LIN {X 0,Y 80.143,Z 462.652,A -85,B 0,C 180,E1 -28635.283,E2 -28635.283} C_VEL
LIN {X 0,Y 70.616,Z 465.452,A -85,B 0,C 180,E1 -28643.46,E2 -28643.46} C_VEL
LIN {X 0,Y 62.833,Z 466.653,A -85,B 0,C 180,E1 -28654.005,E2 -28654.005} C_VEL
LIN {X 0,Y 57.253,Z 466.196,A -85,B 0,C 180,E1 -28667.437,E2 -28667.437} C_VEL
LIN {X 0,Y 55.104,Z 464.603,A -85,B 0,C 180,E1 -28679.324,E2 -28679.324} C_VEL
LIN {X 0,Y 55.173,Z 461.919,A -85,B 0,C 180,E1 -28691.43,E2 -28691.43} C_VEL
LIN {X 0,Y 57.247,Z 458.084,A -85,B 0,C 180,E1 -28702.947,E2 -28702.947} C_VEL
LIN {X 0,Y 60.792,Z 453.051,A -85,B 0,C 180,E1 -28713.313,E2 -28713.313} C_VEL
LIN {X 0,Y 65.825,Z 446.657,A -85,B 0,C 180,E1 -28722.329,E2 -28722.329} C_VEL
LIN {X 0,Y 72.033,Z 438.683,A -85,B 0,C 180,E1 -28729.966,E2 -28729.966} C_VEL
LIN {X 0,Y 78.078,Z 430.306,A -85,B 0,C 180,E1 -28735.419,E2 -28735.419} C_VEL
LIN {X 0,Y 84.431,Z 420.35,A -85,B 0,C 180,E1 -28739.962,E2 -28739.962} C_VEL
LIN {X 0,Y 90.728,Z 408.912,A -85,B 0,C 180,E1 -28743.564,E2 -28743.564} C_VEL
LIN {X 0,Y 96.097,Z 396.85,A -85,B 0,C 180,E1 -28746.199,E2 -28746.199} C_VEL
LIN {X 0,Y 100.408,Z 384.592,A -85,B 0,C 180,E1 -28748.083,E2 -28748.083} C_VEL
LIN {X 0,Y 103.626,Z 371.826,A -85,B 0,C 180,E1 -28749.475,E2 -28749.475} C_VEL
LIN {X 0,Y 105.918,Z 358.431,A -85,B 0,C 180,E1 -28750.304,E2 -28750.304} C_VEL
LIN {X 0,Y 108.067,Z 338.734,A -85,B 0,C 180,E1 -28751.162,E2 -28751.162} C_VEL
LIN {X 0,Y 104.341,Z 329.904,A -85,B 0,C 180,E1 -28755.707,E2 -28755.707} C_VEL
LIN {X 0,Y 101.007,Z 322.981,A -85,B 0,C 180,E1 -28760.449,E2 -28760.449} C_VEL
LIN {X 0,Y 97.749,Z 316.809,A -85,B 0,C 180,E1 -28766.34,E2 -28766.34} C_VEL
LIN {X 0,Y 95.442,Z 312.81,A -85,B 0,C 180,E1 -28771.912,E2 -28771.912} C_VEL
LIN {X 0,Y 93.603,Z 309.407,A -85,B 0,C 180,E1 -28779.127,E2 -28779.127} C_VEL
LIN {X 0,Y 93.461,Z 308.73,A -85,B 0,C 180,E1 -28780.263,E2 -28780.263} C_VEL
LIN {X 0,Y 92.946,Z 308.181,A -85,B 0,C 180,E1 -28789.407,E2 -28789.407} C_VEL
LIN {X 0,Y 93.809,Z 308.628,A -85,B 0,C 180,E1 -28795.889,E2 -28795.889} C_VEL
LIN {X 0,Y 95.125,Z 311.836,A -85,B 0,C 180,E1 -28801.581,E2 -28801.581} C_VEL
LIN {X 0,Y 95.941,Z 313.158,A -85,B 0,C 180,E1 -28803.928,E2 -28803.928} C_VEL
LIN {X 0,Y 98.143,Z 317.367,A -85,B 0,C 180,E1 -28809.012,E2 -28809.012} C_VEL
LIN {X 0,Y 100.767,Z 322.371,A -85,B 0,C 180,E1 -28813.745,E2 -28813.745} C_VEL
LIN {X 0,Y 103.793,Z 328.796,A -85,B 0,C 180,E1 -28818.18,E2 -28818.18} C_VEL
LIN {X 0,Y 105.853,Z 333.789,A -85,B 0,C 180,E1 -28820.892,E2 -28820.892} C_VEL
LIN {X 0,Y 107.916,Z 341.39,A -85,B 0,C 180,E1 -28823.662,E2 -28823.662} C_VEL
LIN {X 0,Y 104.902,Z 367.889,A -85,B 0,C 180,E1 -28824.956,E2 -28824.956} C_VEL
LIN {X 0,Y 102.032,Z 381.003,A -85,B 0,C 180,E1 -28825.912,E2 -28825.912} C_VEL
LIN {X 0,Y 98.4,Z 392.975,A -85,B 0,C 180,E1 -28827.34,E2 -28827.34} C_VEL
LIN {X 0,Y 93.689,Z 404.682,A -85,B 0,C 180,E1 -28829.305,E2 -28829.305} C_VEL
LIN {X 0,Y 88.116,Z 416.043,A -85,B 0,C 180,E1 -28832.068,E2 -28832.068} C_VEL
LIN {X 0,Y 82.155,Z 426.308,A -85,B 0,C 180,E1 -28835.643,E2 -28835.643} C_VEL
LIN {X 0,Y 75.809,Z 435.686,A -85,B 0,C 180,E1 -28840.318,E2 -28840.318} C_VEL
LIN {X 0,Y 69.304,Z 444.511,A -85,B 0,C 180,E1 -28846.805,E2 -28846.805} C_VEL
LIN {X 0,Y 63.686,Z 451.702,A -85,B 0,C 180,E1 -28854.596,E2 -28854.596} C_VEL
LIN {X 0,Y 58.752,Z 458.213,A -85,B 0,C 180,E1 -28865.25,E2 -28865.25} C_VEL
LIN {X 0,Y 56.338,Z 462.494,A -85,B 0,C 180,E1 -28875.554,E2 -28875.554} C_VEL
LIN {X 0,Y 55.593,Z 464.74,A -85,B 0,C 180,E1 -28882.738,E2 -28882.738} C_VEL
LIN {X 0,Y 55.575,Z 466.509,A -85,B 0,C 180,E1 -28890.001,E2 -28890.001} C_VEL
LIN {X 0,Y 55.608,Z 467.791,A -85,B 0,C 180,E1 -28897.262,E2 -28897.262} C_VEL
LIN {X 0,Y 57.825,Z 469.197,A -85,B 0,C 180,E1 -28911.385,E2 -28911.385} C_VEL
LIN {X 0,Y 60.051,Z 469.337,A -85,B 0,C 180,E1 -28917.914,E2 -28917.914} C_VEL
LIN {X 0,Y 66.681,Z 468.446,A -85,B 0,C 180,E1 -28929.227,E2 -28929.227} C_VEL
LIN {X 0,Y 75.465,Z 466.073,A -85,B 0,C 180,E1 -28938.163,E2 -28938.163} C_VEL
LIN {X 0,Y 84.713,Z 462.524,A -85,B 0,C 180,E1 -28944.498,E2 -28944.498} C_VEL
LIN {X 0,Y 94.027,Z 457.924,A -85,B 0,C 180,E1 -28949.268,E2 -28949.268} C_VEL
LIN {X 0,Y 104.37,Z 451.684,A -85,B 0,C 180,E1 -28953.154,E2 -28953.154} C_VEL
LIN {X 0,Y 113.627,Z 444.931,A -85,B 0,C 180,E1 -28955.827,E2 -28955.827} C_VEL
LIN {X 0,Y 121.391,Z 438.132,A -85,B 0,C 180,E1 -28957.87,E2 -28957.87} C_VEL
LIN {X 0,Y 129.468,Z 429.934,A -85,B 0,C 180,E1 -28959.455,E2 -28959.455} C_VEL
LIN {X 0,Y 137.598,Z 419.98,A -85,B 0,C 180,E1 -28960.894,E2 -28960.894} C_VEL
LIN {X 0,Y 144.987,Z 408.845,A -85,B 0,C 180,E1 -28962.043,E2 -28962.043} C_VEL
LIN {X 0,Y 151.3,Z 396.986,A -85,B 0,C 180,E1 -28962.906,E2 -28962.906} C_VEL
LIN {X 0,Y 156.326,Z 384.653,A -85,B 0,C 180,E1 -28963.497,E2 -28963.497} C_VEL
LIN {X 0,Y 158.733,Z 376.969,A -85,B 0,C 180,E1 -28963.857,E2 -28963.857} C_VEL
LIN {X 0,Y 158.771,Z 375.715,A -85,B 0,C 180,E1 -28965.805,E2 -28965.805} C_VEL
LIN {X 0,Y 158.9,Z 375.659,A -85,B 0,C 180,E1 -28970.925,E2 -28970.925} C_VEL
LIN {X 0,Y 158.875,Z 376.131,A -85,B 0,C 180,E1 -28971.572,E2 -28971.572} C_VEL
LIN {X 0,Y 154.358,Z 389.482,A -85,B 0,C 180,E1 -28972.268,E2 -28972.268} C_VEL
LIN {X 0,Y 148.655,Z 401.811,A -85,B 0,C 180,E1 -28973.132,E2 -28973.132} C_VEL
LIN {X 0,Y 141.614,Z 413.626,A -85,B 0,C 180,E1 -28974.304,E2 -28974.304} C_VEL
LIN {X 0,Y 133.905,Z 424.057,A -85,B 0,C 180,E1 -28975.723,E2 -28975.723} C_VEL
LIN {X 0,Y 133.572,Z 424.448,A -85,B 0,C 180,E1 -28975.789,E2 -28975.789} C_VEL
LIN {X 0,Y 129.671,Z 428.845,A -85,B 0,C 180,E1 -28976.27,E2 -28976.27} C_VEL
LIN {X 0,Y 122.489,Z 435.757,A -85,B 0,C 180,E1 -28976.372,E2 -28976.372} C_VEL
LIN {X 0,Y 114.892,Z 441.999,A -85,B 0,C 180,E1 -28976.58,E2 -28976.58} C_VEL
LIN {X 0,Y 110.361,Z 445.395,A -85,B 0,C 180,E1 -28977.313,E2 -28977.313} C_VEL
LIN {X 0,Y 100.78,Z 451.794,A -85,B 0,C 180,E1 -28980,E2 -28980} C_VEL
LIN {X 0,Y 91.515,Z 456.863,A -85,B 0,C 180,E1 -28983.289,E2 -28983.289} C_VEL
LIN {X 0,Y 81.576,Z 461.185,A -85,B 0,C 180,E1 -28987.791,E2 -28987.791} C_VEL
LIN {X 0,Y 72.299,Z 464.234,A -85,B 0,C 180,E1 -28993.57,E2 -28993.57} C_VEL
LIN {X 0,Y 66.343,Z 465.673,A -85,B 0,C 180,E1 -28998.531,E2 -28998.531} C_VEL
LIN {X 0,Y 61.441,Z 466.514,A -85,B 0,C 180,E1 -29003.779,E2 -29003.779} C_VEL
LIN {X 0,Y 56.929,Z 466.878,A -85,B 0,C 180,E1 -29010.211,E2 -29010.211} C_VEL
LIN {X 0,Y 50.934,Z 466.399,A -85,B 0,C 180,E1 -29023.625,E2 -29023.625} C_VEL
LIN {X 0,Y 48.512,Z 465.135,A -85,B 0,C 180,E1 -29034.585,E2 -29034.585} C_VEL
LIN {X 0,Y 47.86,Z 462.636,A -85,B 0,C 180,E1 -29048.461,E2 -29048.461} C_VEL
LIN {X 0,Y 49.685,Z 458.979,A -85,B 0,C 180,E1 -29061.964,E2 -29061.964} C_VEL
LIN {X 0,Y 53.281,Z 454.221,A -85,B 0,C 180,E1 -29073.78,E2 -29073.78} C_VEL
LIN {X 0,Y 58.537,Z 448.091,A -85,B 0,C 180,E1 -29083.892,E2 -29083.892} C_VEL
LIN {X 0,Y 65.081,Z 440.379,A -85,B 0,C 180,E1 -29092.206,E2 -29092.206} C_VEL
LIN {X 0,Y 71.853,Z 431.804,A -85,B 0,C 180,E1 -29098.32,E2 -29098.32} C_VEL
LIN {X 0,Y 78.079,Z 422.9,A -85,B 0,C 180,E1 -29102.687,E2 -29102.687} C_VEL
LIN {X 0,Y 84.591,Z 412.105,A -85,B 0,C 180,E1 -29106.295,E2 -29106.295} C_VEL
LIN {X 0,Y 89.767,Z 401.767,A -85,B 0,C 180,E1 -29108.779,E2 -29108.779} C_VEL
LIN {X 0,Y 94.457,Z 390.338,A -85,B 0,C 180,E1 -29110.725,E2 -29110.725} C_VEL
LIN {X 0,Y 98.345,Z 377.738,A -85,B 0,C 180,E1 -29112.265,E2 -29112.265} C_VEL
LIN {X 0,Y 101.146,Z 364.738,A -85,B 0,C 180,E1 -29113.277,E2 -29113.277} C_VEL
LIN {X 0,Y 103.972,Z 342.423,A -85,B 0,C 180,E1 -29114.214,E2 -29114.214} C_VEL
LIN {X 0,Y 103.927,Z 341.351,A -85,B 0,C 180,E1 -29114.413,E2 -29114.413} C_VEL
LIN {X 0,Y 100.809,Z 333.593,A -85,B 0,C 180,E1 -29118.818,E2 -29118.818} C_VEL
LIN {X 0,Y 98.31,Z 328.065,A -85,B 0,C 180,E1 -29123.019,E2 -29123.019} C_VEL
LIN {X 0,Y 95.853,Z 323.069,A -85,B 0,C 180,E1 -29128.081,E2 -29128.081} C_VEL
LIN {X 0,Y 93.967,Z 319.405,A -85,B 0,C 180,E1 -29133.336,E2 -29133.336} C_VEL
LIN {X 0,Y 92.445,Z 316.161,A -85,B 0,C 180,E1 -29140.321,E2 -29140.321} C_VEL
LIN {X 0,Y 92.365,Z 315.681,A -85,B 0,C 180,E1 -29141.153,E2 -29141.153} C_VEL
LIN {X 0,Y 92.138,Z 315.199,A -85,B 0,C 180,E1 -29151.225,E2 -29151.225} C_VEL
LIN {X 0,Y 92.68,Z 315.658,A -85,B 0,C 180,E1 -29155.106,E2 -29155.106} C_VEL
LIN {X 0,Y 94.009,Z 318.884,A -85,B 0,C 180,E1 -29161.2,E2 -29161.2} C_VEL
LIN {X 0,Y 96.115,Z 323.29,A -85,B 0,C 180,E1 -29167.038,E2 -29167.038} C_VEL
LIN {X 0,Y 98.597,Z 328.46,A -85,B 0,C 180,E1 -29172.073,E2 -29172.073} C_VEL
LIN {X 0,Y 101.481,Z 335.268,A -85,B 0,C 180,E1 -29176.804,E2 -29176.804} C_VEL
LIN {X 0,Y 102.716,Z 338.689,A -85,B 0,C 180,E1 -29178.621,E2 -29178.621} C_VEL
LIN {X 0,Y 103.912,Z 343.538,A -85,B 0,C 180,E1 -29180.506,E2 -29180.506} C_VEL
LIN {X 0,Y 101.002,Z 367.826,A -85,B 0,C 180,E1 -29181.66,E2 -29181.66} C_VEL
LIN {X 0,Y 97.988,Z 381.076,A -85,B 0,C 180,E1 -29182.57,E2 -29182.57} C_VEL
LIN {X 0,Y 94.191,Z 393.017,A -85,B 0,C 180,E1 -29183.935,E2 -29183.935} C_VEL
LIN {X 0,Y 88.938,Z 405.481,A -85,B 0,C 180,E1 -29185.992,E2 -29185.992} C_VEL
LIN {X 0,Y 83.084,Z 416.643,A -85,B 0,C 180,E1 -29188.646,E2 -29188.646} C_VEL
LIN {X 0,Y 76.837,Z 426.726,A -85,B 0,C 180,E1 -29192.216,E2 -29192.216} C_VEL
LIN {X 0,Y 69.328,Z 437.039,A -85,B 0,C 180,E1 -29197.587,E2 -29197.587} C_VEL
LIN {X 0,Y 63.138,Z 444.738,A -85,B 0,C 180,E1 -29203.656,E2 -29203.656} C_VEL
LIN {X 0,Y 57.074,Z 451.82,A -85,B 0,C 180,E1 -29212,E2 -29212} C_VEL
LIN {X 0,Y 52.355,Z 457.449,A -85,B 0,C 180,E1 -29221.978,E2 -29221.978} C_VEL
LIN {X 0,Y 49.482,Z 461.86,A -85,B 0,C 180,E1 -29233.499,E2 -29233.499} C_VEL
LIN {X 0,Y 48.563,Z 464.166,A -85,B 0,C 180,E1 -29241.68,E2 -29241.68} C_VEL
LIN {X 0,Y 48.475,Z 466.029,A -85,B 0,C 180,E1 -29250.001,E2 -29250.001} C_VEL
LIN {X 0,Y 48.571,Z 467.389,A -85,B 0,C 180,E1 -29258.321,E2 -29258.321} C_VEL
LIN {X 0,Y 51.257,Z 468.909,A -85,B 0,C 180,E1 -29274.29,E2 -29274.29} C_VEL
LIN {X 0,Y 57.232,Z 468.956,A -85,B 0,C 180,E1 -29287.88,E2 -29287.88} C_VEL
LIN {X 0,Y 65.91,Z 467.458,A -85,B 0,C 180,E1 -29298.282,E2 -29298.282} C_VEL
LIN {X 0,Y 76.282,Z 464.461,A -85,B 0,C 180,E1 -29306.016,E2 -29306.016} C_VEL
LIN {X 0,Y 84.711,Z 461.119,A -85,B 0,C 180,E1 -29310.59,E2 -29310.59} C_VEL
LIN {X 0,Y 93.629,Z 456.771,A -85,B 0,C 180,E1 -29314.258,E2 -29314.258} C_VEL
LIN {X 0,Y 104.528,Z 450.272,A -85,B 0,C 180,E1 -29317.592,E2 -29317.592} C_VEL
LIN {X 0,Y 114.084,Z 443.22,A -85,B 0,C 180,E1 -29319.961,E2 -29319.961} C_VEL
LIN {X 0,Y 122.197,Z 436.141,A -85,B 0,C 180,E1 -29321.618,E2 -29321.618} C_VEL
LIN {X 0,Y 130.495,Z 427.572,A -85,B 0,C 180,E1 -29322.931,E2 -29322.931} C_VEL
LIN {X 0,Y 138.812,Z 417.142,A -85,B 0,C 180,E1 -29324.147,E2 -29324.147} C_VEL
LIN {X 0,Y 145.519,Z 406.849,A -85,B 0,C 180,E1 -29325,E2 -29325} C_VEL
LIN {X 0,Y 151.335,Z 395.752,A -85,B 0,C 180,E1 -29325.655,E2 -29325.655} C_VEL
LIN {X 0,Y 155.998,Z 384.285,A -85,B 0,C 180,E1 -29326.107,E2 -29326.107} C_VEL
LIN {X 0,Y 156.592,Z 382.373,A -85,B 0,C 180,E1 -29326.797,E2 -29326.797} C_VEL
LIN {X 0,Y 156.616,Z 382.279,A -85,B 0,C 180,E1 -29329.179,E2 -29329.179} C_VEL
LIN {X 0,Y 155.615,Z 385.225,A -85,B 0,C 180,E1 -29329.425,E2 -29329.425} C_VEL
LIN {X 0,Y 150.445,Z 397.363,A -85,B 0,C 180,E1 -29330.06,E2 -29330.06} C_VEL
LIN {X 0,Y 144.108,Z 408.888,A -85,B 0,C 180,E1 -29330.958,E2 -29330.958} C_VEL
LIN {X 0,Y 137.312,Z 418.837,A -85,B 0,C 180,E1 -29331.968,E2 -29331.968} C_VEL
LIN {X 0,Y 128.942,Z 428.851,A -85,B 0,C 180,E1 -29333.384,E2 -29333.384} C_VEL
LIN {X 0,Y 119.91,Z 437.68,A -85,B 0,C 180,E1 -29335.125,E2 -29335.125} C_VEL
LIN {X 0,Y 110.361,Z 445.395,A -85,B 0,C 180,E1 -29337.313,E2 -29337.313} C_VEL
LIN {X 0,Y 105.676,Z 448.621,A -85,B 0,C 180,E1 -29338.169,E2 -29338.169} C_VEL
LIN {X 0,Y 97.158,Z 453.545,A -85,B 0,C 180,E1 -29338.872,E2 -29338.872} C_VEL
LIN {X 0,Y 88.334,Z 457.75,A -85,B 0,C 180,E1 -29339.808,E2 -29339.808} C_VEL
LIN {X 0,Y 83.233,Z 459.849,A -85,B 0,C 180,E1 -29341.194,E2 -29341.194} C_VEL
LIN {X 0,Y 73.922,Z 463.134,A -85,B 0,C 180,E1 -29345.456,E2 -29345.456} C_VEL
LIN {X 0,Y 62.604,Z 465.909,A -85,B 0,C 180,E1 -29352.975,E2 -29352.975} C_VEL
LIN {X 0,Y 52.688,Z 467.071,A -85,B 0,C 180,E1 -29363.589,E2 -29363.589} C_VEL
LIN {X 0,Y 48.696,Z 467.057,A -85,B 0,C 180,E1 -29370.007,E2 -29370.007} C_VEL
LIN {X 0,Y 44.917,Z 466.601,A -85,B 0,C 180,E1 -29378.747,E2 -29378.747} C_VEL
LIN {X 0,Y 42.299,Z 465.672,A -85,B 0,C 180,E1 -29388.346,E2 -29388.346} C_VEL
LIN {X 0,Y 40.871,Z 464.188,A -85,B 0,C 180,E1 -29399.293,E2 -29399.293} C_VEL
LIN {X 0,Y 41.311,Z 461.178,A -85,B 0,C 180,E1 -29415.214,E2 -29415.214} C_VEL
LIN {X 0,Y 44.312,Z 456.977,A -85,B 0,C 180,E1 -29429.999,E2 -29429.999} C_VEL
LIN {X 0,Y 49.27,Z 451.55,A -85,B 0,C 180,E1 -29442.357,E2 -29442.357} C_VEL
LIN {X 0,Y 55.77,Z 444.664,A -85,B 0,C 180,E1 -29452.212,E2 -29452.212} C_VEL
LIN {X 0,Y 63.515,Z 436.041,A -85,B 0,C 180,E1 -29459.862,E2 -29459.862} C_VEL
LIN {X 0,Y 70.522,Z 427.194,A -85,B 0,C 180,E1 -29464.96,E2 -29464.96} C_VEL
LIN {X 0,Y 77.204,Z 417.397,A -85,B 0,C 180,E1 -29468.743,E2 -29468.743} C_VEL
LIN {X 0,Y 83.376,Z 406.675,A -85,B 0,C 180,E1 -29471.59,E2 -29471.59} C_VEL
LIN {X 0,Y 88.695,Z 395.35,A -85,B 0,C 180,E1 -29473.712,E2 -29473.712} C_VEL
LIN {X 0,Y 93.048,Z 383.447,A -85,B 0,C 180,E1 -29475.278,E2 -29475.278} C_VEL
LIN {X 0,Y 96.639,Z 369.6,A -85,B 0,C 180,E1 -29476.53,E2 -29476.53} C_VEL
LIN {X 0,Y 98.8,Z 356.665,A -85,B 0,C 180,E1 -29477.181,E2 -29477.181} C_VEL
LIN {X 0,Y 100.189,Z 344.415,A -85,B 0,C 180,E1 -29477.692,E2 -29477.692} C_VEL
LIN {X 0,Y 97.798,Z 338.005,A -85,B 0,C 180,E1 -29481.727,E2 -29481.727} C_VEL
LIN {X 0,Y 95.942,Z 333.572,A -85,B 0,C 180,E1 -29485.39,E2 -29485.39} C_VEL
LIN {X 0,Y 94.106,Z 329.385,A -85,B 0,C 180,E1 -29489.756,E2 -29489.756} C_VEL
LIN {X 0,Y 92.545,Z 325.977,A -85,B 0,C 180,E1 -29494.838,E2 -29494.838} C_VEL
LIN {X 0,Y 91.293,Z 322.624,A -85,B 0,C 180,E1 -29502.065,E2 -29502.065} C_VEL
LIN {X 0,Y 91.181,Z 322.236,A -85,B 0,C 180,E1 -29511.132,E2 -29511.132} C_VEL
LIN {X 0,Y 91.572,Z 322.655,A -85,B 0,C 180,E1 -29514.301,E2 -29514.301} C_VEL
LIN {X 0,Y 92.979,Z 326.399,A -85,B 0,C 180,E1 -29521.213,E2 -29521.213} C_VEL
LIN {X 0,Y 94.616,Z 330.28,A -85,B 0,C 180,E1 -29526.1,E2 -29526.1} C_VEL
LIN {X 0,Y 96.601,Z 334.934,A -85,B 0,C 180,E1 -29530.545,E2 -29530.545} C_VEL
LIN {X 0,Y 98.837,Z 340.828,A -85,B 0,C 180,E1 -29534.733,E2 -29534.733} C_VEL
LIN {X 0,Y 99.727,Z 343.656,A -85,B 0,C 180,E1 -29536.266,E2 -29536.266} C_VEL
LIN {X 0,Y 100.209,Z 345.852,A -85,B 0,C 180,E1 -29537.163,E2 -29537.163} C_VEL
LIN {X 0,Y 97.464,Z 367.498,A -85,B 0,C 180,E1 -29538.116,E2 -29538.116} C_VEL
LIN {X 0,Y 94.289,Z 381.055,A -85,B 0,C 180,E1 -29538.974,E2 -29538.974} C_VEL
LIN {X 0,Y 90.745,Z 391.915,A -85,B 0,C 180,E1 -29540.109,E2 -29540.109} C_VEL
LIN {X 0,Y 86.034,Z 402.977,A -85,B 0,C 180,E1 -29541.692,E2 -29541.692} C_VEL
LIN {X 0,Y 80.693,Z 413.284,A -85,B 0,C 180,E1 -29543.868,E2 -29543.868} C_VEL
LIN {X 0,Y 74.019,Z 423.968,A -85,B 0,C 180,E1 -29547.111,E2 -29547.111} C_VEL
LIN {X 0,Y 67.583,Z 432.684,A -85,B 0,C 180,E1 -29550.919,E2 -29550.919} C_VEL
LIN {X 0,Y 60.919,Z 440.727,A -85,B 0,C 180,E1 -29556.144,E2 -29556.144} C_VEL
LIN {X 0,Y 53.783,Z 448.585,A -85,B 0,C 180,E1 -29564.055,E2 -29564.055} C_VEL
LIN {X 0,Y 47.778,Z 454.83,A -85,B 0,C 180,E1 -29573.959,E2 -29573.959} C_VEL
LIN {X 0,Y 43.639,Z 459.79,A -85,B 0,C 180,E1 -29586.26,E2 -29586.26} C_VEL
LIN {X 0,Y 41.567,Z 463.575,A -85,B 0,C 180,E1 -29600.267,E2 -29600.267} C_VEL
LIN {X 0,Y 41.394,Z 465.501,A -85,B 0,C 180,E1 -29610.002,E2 -29610.002} C_VEL
LIN {X 0,Y 41.569,Z 466.961,A -85,B 0,C 180,E1 -29619.735,E2 -29619.735} C_VEL
LIN {X 0,Y 42.711,Z 467.989,A -85,B 0,C 180,E1 -29629.215,E2 -29629.215} C_VEL
LIN {X 0,Y 47.904,Z 468.887,A -85,B 0,C 180,E1 -29645.934,E2 -29645.934} C_VEL
LIN {X 0,Y 56.384,Z 468.338,A -85,B 0,C 180,E1 -29658.407,E2 -29658.407} C_VEL
LIN {X 0,Y 66.839,Z 466.243,A -85,B 0,C 180,E1 -29667.267,E2 -29667.267} C_VEL
LIN {X 0,Y 78.439,Z 462.604,A -85,B 0,C 180,E1 -29673.636,E2 -29673.636} C_VEL
LIN {X 0,Y 87.637,Z 458.739,A -85,B 0,C 180,E1 -29677.256,E2 -29677.256} C_VEL
LIN {X 0,Y 97.183,Z 453.821,A -85,B 0,C 180,E1 -29680.073,E2 -29680.073} C_VEL
LIN {X 0,Y 106.947,Z 447.702,A -85,B 0,C 180,E1 -29682.34,E2 -29682.34} C_VEL
LIN {X 0,Y 116.826,Z 440.168,A -85,B 0,C 180,E1 -29684.265,E2 -29684.265} C_VEL
LIN {X 0,Y 126.922,Z 430.732,A -85,B 0,C 180,E1 -29685.702,E2 -29685.702} C_VEL
LIN {X 0,Y 135.373,Z 421.088,A -85,B 0,C 180,E1 -29686.76,E2 -29686.76} C_VEL
LIN {X 0,Y 143.014,Z 410.406,A -85,B 0,C 180,E1 -29687.607,E2 -29687.607} C_VEL
LIN {X 0,Y 143.872,Z 409.013,A -85,B 0,C 180,E1 -29687.683,E2 -29687.683} C_VEL
LIN {X 0,Y 143.632,Z 409.371,A -85,B 0,C 180,E1 -29688.13,E2 -29688.13} C_VEL
LIN {X 0,Y 135.987,Z 420.222,A -85,B 0,C 180,E1 -29689.098,E2 -29689.098} C_VEL
LIN {X 0,Y 128.386,Z 429.026,A -85,B 0,C 180,E1 -29690.178,E2 -29690.178} C_VEL
LIN {X 0,Y 118.965,Z 438.019,A -85,B 0,C 180,E1 -29691.701,E2 -29691.701} C_VEL
LIN {X 0,Y 109.64,Z 445.36,A -85,B 0,C 180,E1 -29693.496,E2 -29693.496} C_VEL
LIN {X 0,Y 98.619,Z 452.437,A -85,B 0,C 180,E1 -29696.115,E2 -29696.115} C_VEL
LIN {X 0,Y 88.559,Z 457.574,A -85,B 0,C 180,E1 -29699.202,E2 -29699.202} C_VEL
LIN {X 0,Y 83.233,Z 459.849,A -85,B 0,C 180,E1 -29701.194,E2 -29701.194} C_VEL
LIN {X 0,Y 78.081,Z 461.734,A -85,B 0,C 180,E1 -29702.806,E2 -29702.806} C_VEL
LIN {X 0,Y 68.841,Z 464.344,A -85,B 0,C 180,E1 -29704.786,E2 -29704.786} C_VEL
LIN {X 0,Y 61.398,Z 465.843,A -85,B 0,C 180,E1 -29706.776,E2 -29706.776} C_VEL
LIN {X 0,Y 56.183,Z 466.629,A -85,B 0,C 180,E1 -29709.36,E2 -29709.36} C_VEL
LIN {X 0,Y 54.609,Z 466.765,A -85,B 0,C 180,E1 -29710.564,E2 -29710.564} C_VEL
LIN {X 0,Y 45.22,Z 467.322,A -85,B 0,C 180,E1 -29721.17,E2 -29721.17} C_VEL
LIN {X 0,Y 39.343,Z 466.799,A -85,B 0,C 180,E1 -29732.406,E2 -29732.406} C_VEL
LIN {X 0,Y 34.385,Z 464.848,A -85,B 0,C 180,E1 -29752.178,E2 -29752.178} C_VEL
LIN {X 0,Y 33.828,Z 461.973,A -85,B 0,C 180,E1 -29771.841,E2 -29771.841} C_VEL
LIN {X 0,Y 36.685,Z 457.956,A -85,B 0,C 180,E1 -29789.998,E2 -29789.998} C_VEL
LIN {X 0,Y 41.957,Z 452.734,A -85,B 0,C 180,E1 -29804.55,E2 -29804.55} C_VEL
LIN {X 0,Y 48.992,Z 446.135,A -85,B 0,C 180,E1 -29815.488,E2 -29815.488} C_VEL
LIN {X 0,Y 57.172,Z 437.82,A -85,B 0,C 180,E1 -29823.583,E2 -29823.583} C_VEL
LIN {X 0,Y 64.815,Z 429.013,A -85,B 0,C 180,E1 -29828.859,E2 -29828.859} C_VEL
LIN {X 0,Y 72.363,Z 418.831,A -85,B 0,C 180,E1 -29832.831,E2 -29832.831} C_VEL
LIN {X 0,Y 78.807,Z 408.371,A -85,B 0,C 180,E1 -29835.514,E2 -29835.514} C_VEL
LIN {X 0,Y 84.878,Z 396.18,A -85,B 0,C 180,E1 -29837.676,E2 -29837.676} C_VEL
LIN {X 0,Y 89.536,Z 384.104,A -85,B 0,C 180,E1 -29839.15,E2 -29839.15} C_VEL
LIN {X 0,Y 93.294,Z 370.273,A -85,B 0,C 180,E1 -29840.308,E2 -29840.308} C_VEL
LIN {X 0,Y 95.625,Z 356.92,A -85,B 0,C 180,E1 -29840.922,E2 -29840.922} C_VEL
LIN {X 0,Y 96.743,Z 347.382,A -85,B 0,C 180,E1 -29841.299,E2 -29841.299} C_VEL
LIN {X 0,Y 94.486,Z 340.885,A -85,B 0,C 180,E1 -29846.05,E2 -29846.05} C_VEL
LIN {X 0,Y 92.527,Z 335.889,A -85,B 0,C 180,E1 -29851.233,E2 -29851.233} C_VEL
LIN {X 0,Y 91.191,Z 332.628,A -85,B 0,C 180,E1 -29856.25,E2 -29856.25} C_VEL
LIN {X 0,Y 90.26,Z 329.669,A -85,B 0,C 180,E1 -29862.734,E2 -29862.734} C_VEL
LIN {X 0,Y 90.225,Z 329.274,A -85,B 0,C 180,E1 -29871.037,E2 -29871.037} C_VEL
LIN {X 0,Y 90.473,Z 329.595,A -85,B 0,C 180,E1 -29873.361,E2 -29873.361} C_VEL
LIN {X 0,Y 91.553,Z 332.884,A -85,B 0,C 180,E1 -29879.653,E2 -29879.653} C_VEL
LIN {X 0,Y 93.004,Z 336.85,A -85,B 0,C 180,E1 -29884.721,E2 -29884.721} C_VEL
LIN {X 0,Y 95.06,Z 342.377,A -85,B 0,C 180,E1 -29889.81,E2 -29889.81} C_VEL
LIN {X 0,Y 96.701,Z 347.668,A -85,B 0,C 180,E1 -29893.309,E2 -29893.309} C_VEL
LIN {X 0,Y 96.801,Z 348.151,A -85,B 0,C 180,E1 -29893.534,E2 -29893.534} C_VEL
LIN {X 0,Y 94.148,Z 367.871,A -85,B 0,C 180,E1 -29894.348,E2 -29894.348} C_VEL
LIN {X 0,Y 91.068,Z 380.628,A -85,B 0,C 180,E1 -29895.078,E2 -29895.078} C_VEL
LIN {X 0,Y 86.917,Z 392.766,A -85,B 0,C 180,E1 -29896.223,E2 -29896.223} C_VEL
LIN {X 0,Y 81.267,Z 405.199,A -85,B 0,C 180,E1 -29897.962,E2 -29897.962} C_VEL
LIN {X 0,Y 74.904,Z 416.331,A -85,B 0,C 180,E1 -29900.24,E2 -29900.24} C_VEL
LIN {X 0,Y 68.744,Z 425.396,A -85,B 0,C 180,E1 -29903.062,E2 -29903.062} C_VEL
LIN {X 0,Y 60.973,Z 434.999,A -85,B 0,C 180,E1 -29907.455,E2 -29907.455} C_VEL
LIN {X 0,Y 52.927,Z 443.688,A -85,B 0,C 180,E1 -29913.913,E2 -29913.913} C_VEL
LIN {X 0,Y 45.5,Z 450.926,A -85,B 0,C 180,E1 -29922.805,E2 -29922.805} C_VEL
LIN {X 0,Y 40.332,Z 455.786,A -85,B 0,C 180,E1 -29932.421,E2 -29932.421} C_VEL
LIN {X 0,Y 36.06,Z 460.492,A -85,B 0,C 180,E1 -29947.06,E2 -29947.06} C_VEL
LIN {X 0,Y 34.588,Z 462.982,A -85,B 0,C 180,E1 -29958.278,E2 -29958.278} C_VEL
LIN {X 0,Y 34.296,Z 464.972,A -85,B 0,C 180,E1 -29970.002,E2 -29970.002} C_VEL
LIN {X 0,Y 34.612,Z 466.491,A -85,B 0,C 180,E1 -29981.717,E2 -29981.717} C_VEL
LIN {X 0,Y 36.059,Z 467.608,A -85,B 0,C 180,E1 -29992.944,E2 -29992.944} C_VEL
LIN {X 0,Y 42.336,Z 468.657,A -85,B 0,C 180,E1 -30011.609,E2 -30011.609} C_VEL
LIN {X 0,Y 51.938,Z 468.237,A -85,B 0,C 180,E1 -30024.282,E2 -30024.282} C_VEL
LIN {X 0,Y 57.425,Z 467.482,A -85,B 0,C 180,E1 -30028.949,E2 -30028.949} C_VEL
LIN {X 0,Y 63.284,Z 466.335,A -85,B 0,C 180,E1 -30032.679,E2 -30032.679} C_VEL
LIN {X 0,Y 75.553,Z 462.845,A -85,B 0,C 180,E1 -30038.468,E2 -30038.468} C_VEL
LIN {X 0,Y 85.145,Z 459.145,A -85,B 0,C 180,E1 -30041.665,E2 -30041.665} C_VEL
LIN {X 0,Y 95.012,Z 454.389,A -85,B 0,C 180,E1 -30044.073,E2 -30044.073} C_VEL
LIN {X 0,Y 105.022,Z 448.449,A -85,B 0,C 180,E1 -30046.01,E2 -30046.01} C_VEL
LIN {X 0,Y 115.12,Z 441.13,A -85,B 0,C 180,E1 -30047.633,E2 -30047.633} C_VEL
LIN {X 0,Y 117.03,Z 439.559,A -85,B 0,C 180,E1 -30048.457,E2 -30048.457} C_VEL
LIN {X 0,Y 107.024,Z 446.991,A -85,B 0,C 180,E1 -30050.069,E2 -30050.069} C_VEL
LIN {X 0,Y 95.162,Z 454.006,A -85,B 0,C 180,E1 -30052.478,E2 -30052.478} C_VEL
LIN {X 0,Y 84.62,Z 458.92,A -85,B 0,C 180,E1 -30055.31,E2 -30055.31} C_VEL
LIN {X 0,Y 77.37,Z 461.643,A -85,B 0,C 180,E1 -30057.72,E2 -30057.72} C_VEL
LIN {X 0,Y 70.285,Z 463.784,A -85,B 0,C 180,E1 -30060.662,E2 -30060.662} C_VEL
LIN {X 0,Y 59.497,Z 466.149,A -85,B 0,C 180,E1 -30066.784,E2 -30066.784} C_VEL
LIN {X 0,Y 54.609,Z 466.765,A -85,B 0,C 180,E1 -30070.564,E2 -30070.564} C_VEL
LIN {X 0,Y 49.761,Z 467.244,A -85,B 0,C 180,E1 -30074.252,E2 -30074.252} C_VEL
LIN {X 0,Y 41.066,Z 467.332,A -85,B 0,C 180,E1 -30080.294,E2 -30080.294} C_VEL
LIN {X 0,Y 34.435,Z 466.866,A -85,B 0,C 180,E1 -30086.998,E2 -30086.998} C_VEL
LIN {X 0,Y 30.468,Z 466.147,A -85,B 0,C 180,E1 -30094.722,E2 -30094.722} C_VEL
LIN {X 0,Y 29.505,Z 465.786,A -85,B 0,C 180,E1 -30097.988,E2 -30097.988} C_VEL
LIN {X 0,Y 26.678,Z 463.742,A -85,B 0,C 180,E1 -30118.203,E2 -30118.203} C_VEL
LIN {X 0,Y 28.199,Z 459.78,A -85,B 0,C 180,E1 -30145.513,E2 -30145.513} C_VEL
LIN {X 0,Y 32.574,Z 455.668,A -85,B 0,C 180,E1 -30162.458,E2 -30162.458} C_VEL
LIN {X 0,Y 38.772,Z 450.504,A -85,B 0,C 180,E1 -30174.995,E2 -30174.995} C_VEL
LIN {X 0,Y 46.622,Z 443.719,A -85,B 0,C 180,E1 -30184.421,E2 -30184.421} C_VEL
LIN {X 0,Y 54.266,Z 436.396,A -85,B 0,C 180,E1 -30190.355,E2 -30190.355} C_VEL
LIN {X 0,Y 62.21,Z 427.551,A -85,B 0,C 180,E1 -30194.915,E2 -30194.915} C_VEL
LIN {X 0,Y 69.603,Z 417.762,A -85,B 0,C 180,E1 -30198.13,E2 -30198.13} C_VEL
LIN {X 0,Y 76.452,Z 406.841,A -85,B 0,C 180,E1 -30200.477,E2 -30200.477} C_VEL
LIN {X 0,Y 82.271,Z 395.295,A -85,B 0,C 180,E1 -30202.2,E2 -30202.2} C_VEL
LIN {X 0,Y 86.956,Z 383.167,A -85,B 0,C 180,E1 -30203.433,E2 -30203.433} C_VEL
LIN {X 0,Y 90.625,Z 369.826,A -85,B 0,C 180,E1 -30204.391,E2 -30204.391} C_VEL
LIN {X 0,Y 92.877,Z 357.086,A -85,B 0,C 180,E1 -30204.888,E2 -30204.888} C_VEL
LIN {X 0,Y 93.639,Z 350.576,A -85,B 0,C 180,E1 -30205.166,E2 -30205.166} C_VEL
LIN {X 0,Y 92.144,Z 345.871,A -85,B 0,C 180,E1 -30209.042,E2 -30209.042} C_VEL
LIN {X 0,Y 90.856,Z 341.987,A -85,B 0,C 180,E1 -30213.338,E2 -30213.338} C_VEL
LIN {X 0,Y 89.865,Z 339.195,A -85,B 0,C 180,E1 -30217.82,E2 -30217.82} C_VEL
LIN {X 0,Y 89.205,Z 336.55,A -85,B 0,C 180,E1 -30224.091,E2 -30224.091} C_VEL
LIN {X 0,Y 89.382,Z 336.391,A -85,B 0,C 180,E1 -30232.117,E2 -30232.117} C_VEL
LIN {X 0,Y 90.24,Z 339.597,A -85,B 0,C 180,E1 -30238.326,E2 -30238.326} C_VEL
LIN {X 0,Y 91.619,Z 343.91,A -85,B 0,C 180,E1 -30243.851,E2 -30243.851} C_VEL
LIN {X 0,Y 93.365,Z 349.699,A -85,B 0,C 180,E1 -30248.771,E2 -30248.771} C_VEL
LIN {X 0,Y 93.75,Z 351.04,A -85,B 0,C 180,E1 -30249.702,E2 -30249.702} C_VEL
LIN {X 0,Y 91.145,Z 368.922,A -85,B 0,C 180,E1 -30250.365,E2 -30250.365} C_VEL
LIN {X 0,Y 87.757,Z 381.973,A -85,B 0,C 180,E1 -30251.036,E2 -30251.036} C_VEL
LIN {X 0,Y 83.524,Z 393.57,A -85,B 0,C 180,E1 -30251.998,E2 -30251.998} C_VEL
LIN {X 0,Y 77.704,Z 405.806,A -85,B 0,C 180,E1 -30253.524,E2 -30253.524} C_VEL
LIN {X 0,Y 71.113,Z 416.749,A -85,B 0,C 180,E1 -30255.515,E2 -30255.515} C_VEL
LIN {X 0,Y 64.667,Z 425.693,A -85,B 0,C 180,E1 -30258.025,E2 -30258.025} C_VEL
LIN {X 0,Y 57.287,Z 434.342,A -85,B 0,C 180,E1 -30261.594,E2 -30261.594} C_VEL
LIN {X 0,Y 49.304,Z 442.45,A -85,B 0,C 180,E1 -30267.017,E2 -30267.017} C_VEL
LIN {X 0,Y 41.002,Z 449.874,A -85,B 0,C 180,E1 -30275.496,E2 -30275.496} C_VEL
LIN {X 0,Y 34.942,Z 454.882,A -85,B 0,C 180,E1 -30285.257,E2 -30285.257} C_VEL
LIN {X 0,Y 29.628,Z 459.735,A -85,B 0,C 180,E1 -30301.682,E2 -30301.682} C_VEL
LIN {X 0,Y 27.226,Z 463.419,A -85,B 0,C 180,E1 -30322.587,E2 -30322.587} C_VEL
LIN {X 0,Y 27.213,Z 464.422,A -85,B 0,C 180,E1 -30330.002,E2 -30330.002} C_VEL
LIN {X 0,Y 27.699,Z 466.004,A -85,B 0,C 180,E1 -30344.7,E2 -30344.7} C_VEL
LIN {X 0,Y 32.951,Z 467.994,A -85,B 0,C 180,E1 -30369.783,E2 -30369.783} C_VEL
LIN {X 0,Y 37.306,Z 468.424,A -85,B 0,C 180,E1 -30378.901,E2 -30378.901} C_VEL
LIN {X 0,Y 48.129,Z 468.137,A -85,B 0,C 180,E1 -30391.184,E2 -30391.184} C_VEL
LIN {X 0,Y 60.35,Z 466.401,A -85,B 0,C 180,E1 -30398.693,E2 -30398.693} C_VEL
LIN {X 0,Y 68.846,Z 464.385,A -85,B 0,C 180,E1 -30402.167,E2 -30402.167} C_VEL
LIN {X 0,Y 79.852,Z 460.835,A -85,B 0,C 180,E1 -30405.501,E2 -30405.501} C_VEL
LIN {X 0,Y 89.926,Z 456.597,A -85,B 0,C 180,E1 -30407.667,E2 -30407.667} C_VEL
LIN {X 0,Y 93.323,Z 454.958,A -85,B 0,C 180,E1 -30408.239,E2 -30408.239} C_VEL
LIN {X 0,Y 80.983,Z 460.242,A -85,B 0,C 180,E1 -30411.073,E2 -30411.073} C_VEL
LIN {X 0,Y 70.253,Z 463.651,A -85,B 0,C 180,E1 -30414.259,E2 -30414.259} C_VEL
LIN {X 0,Y 63.343,Z 465.289,A -85,B 0,C 180,E1 -30416.944,E2 -30416.944} C_VEL
LIN {X 0,Y 56.227,Z 466.548,A -85,B 0,C 180,E1 -30420.521,E2 -30420.521} C_VEL
LIN {X 0,Y 45.006,Z 467.494,A -85,B 0,C 180,E1 -30428.985,E2 -30428.985} C_VEL
LIN {X 0,Y 34.336,Z 466.992,A -85,B 0,C 180,E1 -30444.166,E2 -30444.166} C_VEL
LIN {X 0,Y 29.505,Z 465.786,A -85,B 0,C 180,E1 -30457.988,E2 -30457.988} C_VEL
LIN {X 0,Y 26.855,Z 464.76,A -85,B 0,C 180,E1 -30468.525,E2 -30468.525} C_VEL
LIN {X 0,Y 23.026,Z 462.373,A -85,B 0,C 180,E1 -30488.956,E2 -30488.956} C_VEL
LIN {X 0,Y 22.246,Z 459.919,A -85,B 0,C 180,E1 -30508.227,E2 -30508.227} C_VEL
LIN {X 0,Y 23.875,Z 457.743,A -85,B 0,C 180,E1 -30521.496,E2 -30521.496} C_VEL
LIN {X 0,Y 24.866,Z 456.947,A -85,B 0,C 180,E1 -30525.142,E2 -30525.142} C_VEL
LIN {X 0,Y 33.247,Z 450.896,A -85,B 0,C 180,E1 -30542.266,E2 -30542.266} C_VEL
LIN {X 0,Y 42.269,Z 443.862,A -85,B 0,C 180,E1 -30551.685,E2 -30551.685} C_VEL
LIN {X 0,Y 51.133,Z 435.913,A -85,B 0,C 180,E1 -30557.306,E2 -30557.306} C_VEL
LIN {X 0,Y 59.743,Z 426.641,A -85,B 0,C 180,E1 -30561.198,E2 -30561.198} C_VEL
LIN {X 0,Y 67.484,Z 416.623,A -85,B 0,C 180,E1 -30563.812,E2 -30563.812} C_VEL
LIN {X 0,Y 74.38,Z 405.788,A -85,B 0,C 180,E1 -30565.616,E2 -30565.616} C_VEL
LIN {X 0,Y 80.582,Z 393.305,A -85,B 0,C 180,E1 -30567.08,E2 -30567.08} C_VEL
LIN {X 0,Y 85.348,Z 380.62,A -85,B 0,C 180,E1 -30568.073,E2 -30568.073} C_VEL
LIN {X 0,Y 88.741,Z 367.749,A -85,B 0,C 180,E1 -30568.746,E2 -30568.746} C_VEL
LIN {X 0,Y 90.937,Z 354.052,A -85,B 0,C 180,E1 -30569.161,E2 -30569.161} C_VEL
LIN {X 0,Y 89.678,Z 349.384,A -85,B 0,C 180,E1 -30573.793,E2 -30573.793} C_VEL
LIN {X 0,Y 88.684,Z 346.014,A -85,B 0,C 180,E1 -30578.91,E2 -30578.91} C_VEL
LIN {X 0,Y 88.229,Z 343.546,A -85,B 0,C 180,E1 -30584.596,E2 -30584.596} C_VEL
LIN {X 0,Y 88.36,Z 343.412,A -85,B 0,C 180,E1 -30591.436,E2 -30591.436} C_VEL
LIN {X 0,Y 88.929,Z 346.188,A -85,B 0,C 180,E1 -30596.817,E2 -30596.817} C_VEL
LIN {X 0,Y 89.914,Z 349.92,A -85,B 0,C 180,E1 -30601.699,E2 -30601.699} C_VEL
LIN {X 0,Y 90.99,Z 354.203,A -85,B 0,C 180,E1 -30605.593,E2 -30605.593} C_VEL
LIN {X 0,Y 88.627,Z 369.423,A -85,B 0,C 180,E1 -30606.13,E2 -30606.13} C_VEL
LIN {X 0,Y 85.343,Z 381.689,A -85,B 0,C 180,E1 -30606.634,E2 -30606.634} C_VEL
LIN {X 0,Y 80.621,Z 394.177,A -85,B 0,C 180,E1 -30607.441,E2 -30607.441} C_VEL
LIN {X 0,Y 74.65,Z 406.266,A -85,B 0,C 180,E1 -30608.696,E2 -30608.696} C_VEL
LIN {X 0,Y 67.858,Z 417.042,A -85,B 0,C 180,E1 -30610.299,E2 -30610.299} C_VEL
LIN {X 0,Y 61.157,Z 425.901,A -85,B 0,C 180,E1 -30612.372,E2 -30612.372} C_VEL
LIN {X 0,Y 52.545,Z 435.376,A -85,B 0,C 180,E1 -30615.813,E2 -30615.813} C_VEL
LIN {X 0,Y 43.354,Z 443.897,A -85,B 0,C 180,E1 -30621.237,E2 -30621.237} C_VEL
LIN {X 0,Y 34.414,Z 450.986,A -85,B 0,C 180,E1 -30629.786,E2 -30629.786} C_VEL
LIN {X 0,Y 25.543,Z 457.428,A -85,B 0,C 180,E1 -30646.544,E2 -30646.544} C_VEL
LIN {X 0,Y 20.877,Z 461.644,A -85,B 0,C 180,E1 -30670.332,E2 -30670.332} C_VEL
LIN {X 0,Y 20.142,Z 463.851,A -85,B 0,C 180,E1 -30690.003,E2 -30690.003} C_VEL
LIN {X 0,Y 20.901,Z 465.517,A -85,B 0,C 180,E1 -30709.652,E2 -30709.652} C_VEL
LIN {X 0,Y 27.856,Z 467.632,A -85,B 0,C 180,E1 -30739.193,E2 -30739.193} C_VEL
LIN {X 0,Y 38.918,Z 468.288,A -85,B 0,C 180,E1 -30754.548,E2 -30754.548} C_VEL
LIN {X 0,Y 51.55,Z 467.425,A -85,B 0,C 180,E1 -30762.619,E2 -30762.619} C_VEL
LIN {X 0,Y 64.824,Z 465.092,A -85,B 0,C 180,E1 -30767.361,E2 -30767.361} C_VEL
LIN {X 0,Y 65.991,Z 464.832,A -85,B 0,C 180,E1 -30767.702,E2 -30767.702} C_VEL
LIN {X 0,Y 66.898,Z 464.566,A -85,B 0,C 180,E1 -30769.015,E2 -30769.015} C_VEL
LIN {X 0,Y 55.725,Z 466.653,A -85,B 0,C 180,E1 -30772.755,E2 -30772.755} C_VEL
LIN {X 0,Y 49.334,Z 467.366,A -85,B 0,C 180,E1 -30775.729,E2 -30775.729} C_VEL
LIN {X 0,Y 42.169,Z 467.714,A -85,B 0,C 180,E1 -30780.251,E2 -30780.251} C_VEL
LIN {X 0,Y 30.287,Z 467.181,A -85,B 0,C 180,E1 -30793.419,E2 -30793.419} C_VEL
LIN {X 0,Y 23.308,Z 465.731,A -85,B 0,C 180,E1 -30810.404,E2 -30810.404} C_VEL
LIN {X 0,Y 19.578,Z 463.43,A -85,B 0,C 180,E1 -30837.417,E2 -30837.417} C_VEL
LIN {X 0,Y 21.341,Z 459.785,A -85,B 0,C 180,E1 -30869.997,E2 -30869.997} C_VEL
LIN {X 0,Y 24.866,Z 456.947,A -85,B 0,C 180,E1 -30885.142,E2 -30885.142} C_VEL
LIN {X 0,Y 27.852,Z 454.486,A -85,B 0,C 180,E1 -30894.869,E2 -30894.869} C_VEL
LIN {X 0,Y 32.562,Z 449.852,A -85,B 0,C 180,E1 -30909.014,E2 -30909.014} C_VEL
LIN {X 0,Y 38.288,Z 444.56,A -85,B 0,C 180,E1 -30919.12,E2 -30919.12} C_VEL
LIN {X 0,Y 42.47,Z 440.989,A -85,B 0,C 180,E1 -30922.4,E2 -30922.4} C_VEL
LIN {X 0,Y 50.966,Z 433.297,A -85,B 0,C 180,E1 -30925.827,E2 -30925.827} C_VEL
LIN {X 0,Y 59.826,Z 423.663,A -85,B 0,C 180,E1 -30928.393,E2 -30928.393} C_VEL
LIN {X 0,Y 68.148,Z 412.423,A -85,B 0,C 180,E1 -30930.175,E2 -30930.175} C_VEL
LIN {X 0,Y 75.034,Z 400.791,A -85,B 0,C 180,E1 -30931.412,E2 -30931.412} C_VEL
LIN {X 0,Y 80.219,Z 389.576,A -85,B 0,C 180,E1 -30932.218,E2 -30932.218} C_VEL
LIN {X 0,Y 84.715,Z 376.426,A -85,B 0,C 180,E1 -30932.938,E2 -30932.938} C_VEL
LIN {X 0,Y 87.856,Z 362.894,A -85,B 0,C 180,E1 -30933.336,E2 -30933.336} C_VEL
LIN {X 0,Y 88.651,Z 357.745,A -85,B 0,C 180,E1 -30933.434,E2 -30933.434} C_VEL
LIN {X 0,Y 87.908,Z 354.515,A -85,B 0,C 180,E1 -30937.311,E2 -30937.311} C_VEL
LIN {X 0,Y 87.438,Z 352.472,A -85,B 0,C 180,E1 -30940.882,E2 -30940.882} C_VEL
LIN {X 0,Y 87.239,Z 350.472,A -85,B 0,C 180,E1 -30946.014,E2 -30946.014} C_VEL
LIN {X 0,Y 87.353,Z 350.6,A -85,B 0,C 180,E1 -30951.039,E2 -30951.039} C_VEL
LIN {X 0,Y 87.745,Z 353.135,A -85,B 0,C 180,E1 -30955.797,E2 -30955.797} C_VEL
LIN {X 0,Y 88.46,Z 356.577,A -85,B 0,C 180,E1 -30960.142,E2 -30960.142} C_VEL
LIN {X 0,Y 88.684,Z 357.723,A -85,B 0,C 180,E1 -30961.276,E2 -30961.276} C_VEL
LIN {X 0,Y 86.492,Z 370.455,A -85,B 0,C 180,E1 -30961.708,E2 -30961.708} C_VEL
LIN {X 0,Y 82.485,Z 384.232,A -85,B 0,C 180,E1 -30962.09,E2 -30962.09} C_VEL
LIN {X 0,Y 77.391,Z 396.722,A -85,B 0,C 180,E1 -30962.686,E2 -30962.686} C_VEL
LIN {X 0,Y 71.299,Z 408.128,A -85,B 0,C 180,E1 -30963.617,E2 -30963.617} C_VEL
LIN {X 0,Y 64.353,Z 418.516,A -85,B 0,C 180,E1 -30964.782,E2 -30964.782} C_VEL
LIN {X 0,Y 56.587,Z 428.068,A -85,B 0,C 180,E1 -30966.51,E2 -30966.51} C_VEL
LIN {X 0,Y 48.039,Z 436.784,A -85,B 0,C 180,E1 -30969.078,E2 -30969.078} C_VEL
LIN {X 0,Y 37.991,Z 445.239,A -85,B 0,C 180,E1 -30973.792,E2 -30973.792} C_VEL
LIN {X 0,Y 28.313,Z 452.003,A -85,B 0,C 180,E1 -30981.44,E2 -30981.44} C_VEL
LIN {X 0,Y 18.368,Z 458.189,A -85,B 0,C 180,E1 -31000.077,E2 -31000.077} C_VEL
LIN {X 0,Y 13.306,Z 462.164,A -85,B 0,C 180,E1 -31034.692,E2 -31034.692} C_VEL
LIN {X 0,Y 13.06,Z 463.219,A -85,B 0,C 180,E1 -31050.005,E2 -31050.005} C_VEL
LIN {X 0,Y 14.416,Z 464.991,A -85,B 0,C 180,E1 -31079.182,E2 -31079.182} C_VEL
LIN {X 0,Y 18.402,Z 466.327,A -85,B 0,C 180,E1 -31099.81,E2 -31099.81} C_VEL
LIN {X 0,Y 29.931,Z 467.838,A -85,B 0,C 180,E1 -31119.925,E2 -31119.925} C_VEL
LIN {X 0,Y 43.105,Z 467.92,A -85,B 0,C 180,E1 -31128.038,E2 -31128.038} C_VEL
LIN {X 0,Y 42.899,Z 467.896,A -85,B 0,C 180,E1 -31129.413,E2 -31129.413} C_VEL
LIN {X 0,Y 35.376,Z 467.879,A -85,B 0,C 180,E1 -31133.385,E2 -31133.385} C_VEL
LIN {X 0,Y 27.592,Z 467.366,A -85,B 0,C 180,E1 -31140.001,E2 -31140.001} C_VEL
LIN {X 0,Y 21.349,Z 466.446,A -85,B 0,C 180,E1 -31149.016,E2 -31149.016} C_VEL
LIN {X 0,Y 15.47,Z 464.933,A -85,B 0,C 180,E1 -31167.023,E2 -31167.023} C_VEL
LIN {X 0,Y 12.457,Z 461.914,A -85,B 0,C 180,E1 -31213.61,E2 -31213.61} C_VEL
LIN {X 0,Y 18.031,Z 457.672,A -85,B 0,C 180,E1 -31252.937,E2 -31252.937} C_VEL
LIN {X 0,Y 26.466,Z 452.563,A -85,B 0,C 180,E1 -31269.811,E2 -31269.811} C_VEL
LIN {X 0,Y 35.36,Z 446.564,A -85,B 0,C 180,E1 -31278.184,E2 -31278.184} C_VEL
LIN {X 0,Y 42.47,Z 440.989,A -85,B 0,C 180,E1 -31282.4,E2 -31282.4} C_VEL
LIN {X 0,Y 46.59,Z 437.267,A -85,B 0,C 180,E1 -31285.006,E2 -31285.006} C_VEL
LIN {X 0,Y 52.583,Z 430.758,A -85,B 0,C 180,E1 -31290.2,E2 -31290.2} C_VEL
LIN {X 0,Y 58.318,Z 423.676,A -85,B 0,C 180,E1 -31294.343,E2 -31294.343} C_VEL
LIN {X 0,Y 61.82,Z 419.051,A -85,B 0,C 180,E1 -31295.533,E2 -31295.533} C_VEL
LIN {X 0,Y 69.697,Z 407.547,A -85,B 0,C 180,E1 -31296.361,E2 -31296.361} C_VEL
LIN {X 0,Y 76.332,Z 395.199,A -85,B 0,C 180,E1 -31297.028,E2 -31297.028} C_VEL
LIN {X 0,Y 81.401,Z 382.624,A -85,B 0,C 180,E1 -31297.44,E2 -31297.44} C_VEL
LIN {X 0,Y 85.271,Z 369.039,A -85,B 0,C 180,E1 -31297.832,E2 -31297.832} C_VEL
LIN {X 0,Y 86.682,Z 361.626,A -85,B 0,C 180,E1 -31298.014,E2 -31298.014} C_VEL
LIN {X 0,Y 86.33,Z 359.234,A -85,B 0,C 180,E1 -31302.074,E2 -31302.074} C_VEL
LIN {X 0,Y 86.277,Z 357.655,A -85,B 0,C 180,E1 -31305.855,E2 -31305.855} C_VEL
LIN {X 0,Y 86.352,Z 357.642,A -85,B 0,C 180,E1 -31310.372,E2 -31310.372} C_VEL
LIN {X 0,Y 86.563,Z 360.07,A -85,B 0,C 180,E1 -31314.773,E2 -31314.773} C_VEL
LIN {X 0,Y 86.761,Z 361.661,A -85,B 0,C 180,E1 -31316.841,E2 -31316.841} C_VEL
LIN {X 0,Y 84.143,Z 374.208,A -85,B 0,C 180,E1 -31317.104,E2 -31317.104} C_VEL
LIN {X 0,Y 80.417,Z 385.967,A -85,B 0,C 180,E1 -31317.284,E2 -31317.284} C_VEL
LIN {X 0,Y 74.738,Z 398.912,A -85,B 0,C 180,E1 -31317.578,E2 -31317.578} C_VEL
LIN {X 0,Y 68.56,Z 409.846,A -85,B 0,C 180,E1 -31318.066,E2 -31318.066} C_VEL
LIN {X 0,Y 60.628,Z 421.027,A -85,B 0,C 180,E1 -31318.816,E2 -31318.816} C_VEL
LIN {X 0,Y 52.706,Z 430.054,A -85,B 0,C 180,E1 -31319.716,E2 -31319.716} C_VEL
LIN {X 0,Y 42.183,Z 439.852,A -85,B 0,C 180,E1 -31321.621,E2 -31321.621} C_VEL
LIN {X 0,Y 31.734,Z 447.667,A -85,B 0,C 180,E1 -31324.749,E2 -31324.749} C_VEL
LIN {X 0,Y 21.438,Z 453.888,A -85,B 0,C 180,E1 -31330.445,E2 -31330.445} C_VEL
LIN {X 0,Y 11.706,Z 458.814,A -85,B 0,C 180,E1 -31345.781,E2 -31345.781} C_VEL
LIN {X 0,Y 5.963,Z 462.569,A -85,B 0,C 180,E1 -31410.011,E2 -31410.011} C_VEL
LIN {X 0,Y 8.925,Z 464.415,A -85,B 0,C 180,E1 -31461.96,E2 -31461.96} C_VEL
LIN {X 0,Y 14.848,Z 465.852,A -85,B 0,C 180,E1 -31481.219,E2 -31481.219} C_VEL
LIN {X 0,Y 18.02,Z 466.343,A -85,B 0,C 180,E1 -31490.66,E2 -31490.66} C_VEL
LIN {X 0,Y 7.439,Z 463.763,A -85,B 0,C 180,E1 -31519.11,E2 -31519.11} C_VEL
LIN {X 0,Y 7.529,Z 460.401,A -85,B 0,C 180,E1 -31611.016,E2 -31611.016} C_VEL
LIN {X 0,Y 18.296,Z 455.226,A -85,B 0,C 180,E1 -31640.191,E2 -31640.191} C_VEL
LIN {X 0,Y 29.067,Z 449.023,A -85,B 0,C 180,E1 -31647.801,E2 -31647.801} C_VEL
LIN {X 0,Y 40.538,Z 440.778,A -85,B 0,C 180,E1 -31651.804,E2 -31651.804} C_VEL
LIN {X 0,Y 49.016,Z 433.327,A -85,B 0,C 180,E1 -31653.652,E2 -31653.652} C_VEL
LIN {X 0,Y 58.116,Z 423.645,A -85,B 0,C 180,E1 -31655.089,E2 -31655.089} C_VEL
LIN {X 0,Y 61.82,Z 419.051,A -85,B 0,C 180,E1 -31655.533,E2 -31655.533} C_VEL
LIN {X 0,Y 65.122,Z 414.375,A -85,B 0,C 180,E1 -31656.563,E2 -31656.563} C_VEL
LIN {X 0,Y 71.667,Z 403.071,A -85,B 0,C 180,E1 -31660.449,E2 -31660.449} C_VEL
LIN {X 0,Y 75.064,Z 396.192,A -85,B 0,C 180,E1 -31662.05,E2 -31662.05} C_VEL
LIN {X 0,Y 76.709,Z 392.512,A -85,B 0,C 180,E1 -31662.346,E2 -31662.346} C_VEL
LIN {X 0,Y 81.544,Z 379.796,A -85,B 0,C 180,E1 -31662.482,E2 -31662.482} C_VEL
LIN {X 0,Y 85.033,Z 366.213,A -85,B 0,C 180,E1 -31662.705,E2 -31662.705} C_VEL
LIN {X 0,Y 85.08,Z 365.005,A -85,B 0,C 180,E1 -31665.651,E2 -31665.651} C_VEL
LIN {X 0,Y 85.164,Z 365.141,A -85,B 0,C 180,E1 -31670.796,E2 -31670.796} C_VEL
LIN {X 0,Y 85.109,Z 366.158,A -85,B 0,C 180,E1 -31672.265,E2 -31672.265} C_VEL
LIN {X 0,Y 82.133,Z 378.058,A -85,B 0,C 180,E1 -31672.23,E2 -31672.23} C_VEL
LIN {X 0,Y 77.58,Z 390.774,A -85,B 0,C 180,E1 -31672.224,E2 -31672.224} C_VEL
LIN {X 0,Y 71.829,Z 402.614,A -85,B 0,C 180,E1 -31672.156,E2 -31672.156} C_VEL
LIN {X 0,Y 64.745,Z 414.03,A -85,B 0,C 180,E1 -31672.091,E2 -31672.091} C_VEL
LIN {X 0,Y 56.762,Z 424.374,A -85,B 0,C 180,E1 -31672.096,E2 -31672.096} C_VEL
LIN {X 0,Y 47.236,Z 434.252,A -85,B 0,C 180,E1 -31671.994,E2 -31671.994} C_VEL
LIN {X 0,Y 37.26,Z 442.653,A -85,B 0,C 180,E1 -31671.979,E2 -31671.979} C_VEL
LIN {X 0,Y 26.638,Z 449.876,A -85,B 0,C 180,E1 -31671.615,E2 -31671.615} C_VEL
LIN {X 0,Y 17.791,Z 454.739,A -85,B 0,C 180,E1 -31670.925,E2 -31670.925} C_VEL
LIN {X 0,Y 14.26,Z 456.428,A -85,B 0,C 180,E1 -31670.277,E2 -31670.277} C_VEL
LIN {X 0,Y 14.646,Z 456.215,A -85,B 0,C 180,E1 -31663.666,E2 -31663.666} C_VEL
LIN {X 0,Y 26.246,Z 450.034,A -85,B 0,C 180,E1 -31661.931,E2 -31661.931} C_VEL
LIN {X 0,Y 36.985,Z 442.749,A -85,B 0,C 180,E1 -31661.821,E2 -31661.821} C_VEL
LIN {X 0,Y 47.112,Z 434.224,A -85,B 0,C 180,E1 -31661.929,E2 -31661.929} C_VEL
LIN {X 0,Y 56.33,Z 424.692,A -85,B 0,C 180,E1 -31662.046,E2 -31662.046} C_VEL
LIN {X 0,Y 64.605,Z 414.051,A -85,B 0,C 180,E1 -31662.146,E2 -31662.146} C_VEL
LIN {X 0,Y 71.808,Z 402.444,A -85,B 0,C 180,E1 -31662.251,E2 -31662.251} C_VEL
LIN {X 0,Y 76.709,Z 392.512,A -85,B 0,C 180,E1 -31662.346,E2 -31662.346} C_VEL
LIN {X 0,Y 80.527,Z 393.33,A -85,B 0,C 180,E1 -31662.521,E2 -31662.521} C_VEL
LIN {X 0,Y 80.527,Z 600,A -85,B 0,C 180,E1 -31662.521,E2 -31662.521} C_VEL
LIN {X 0,Y 80.527,Z 600,A -85,B 0,C 180,E1 -31662.521,E2 -31662.521}

QRS_NEXT_CUT()

QRS_NEXT()
QRS_HOME()

END
